REGION Network 49: Phmi Connect
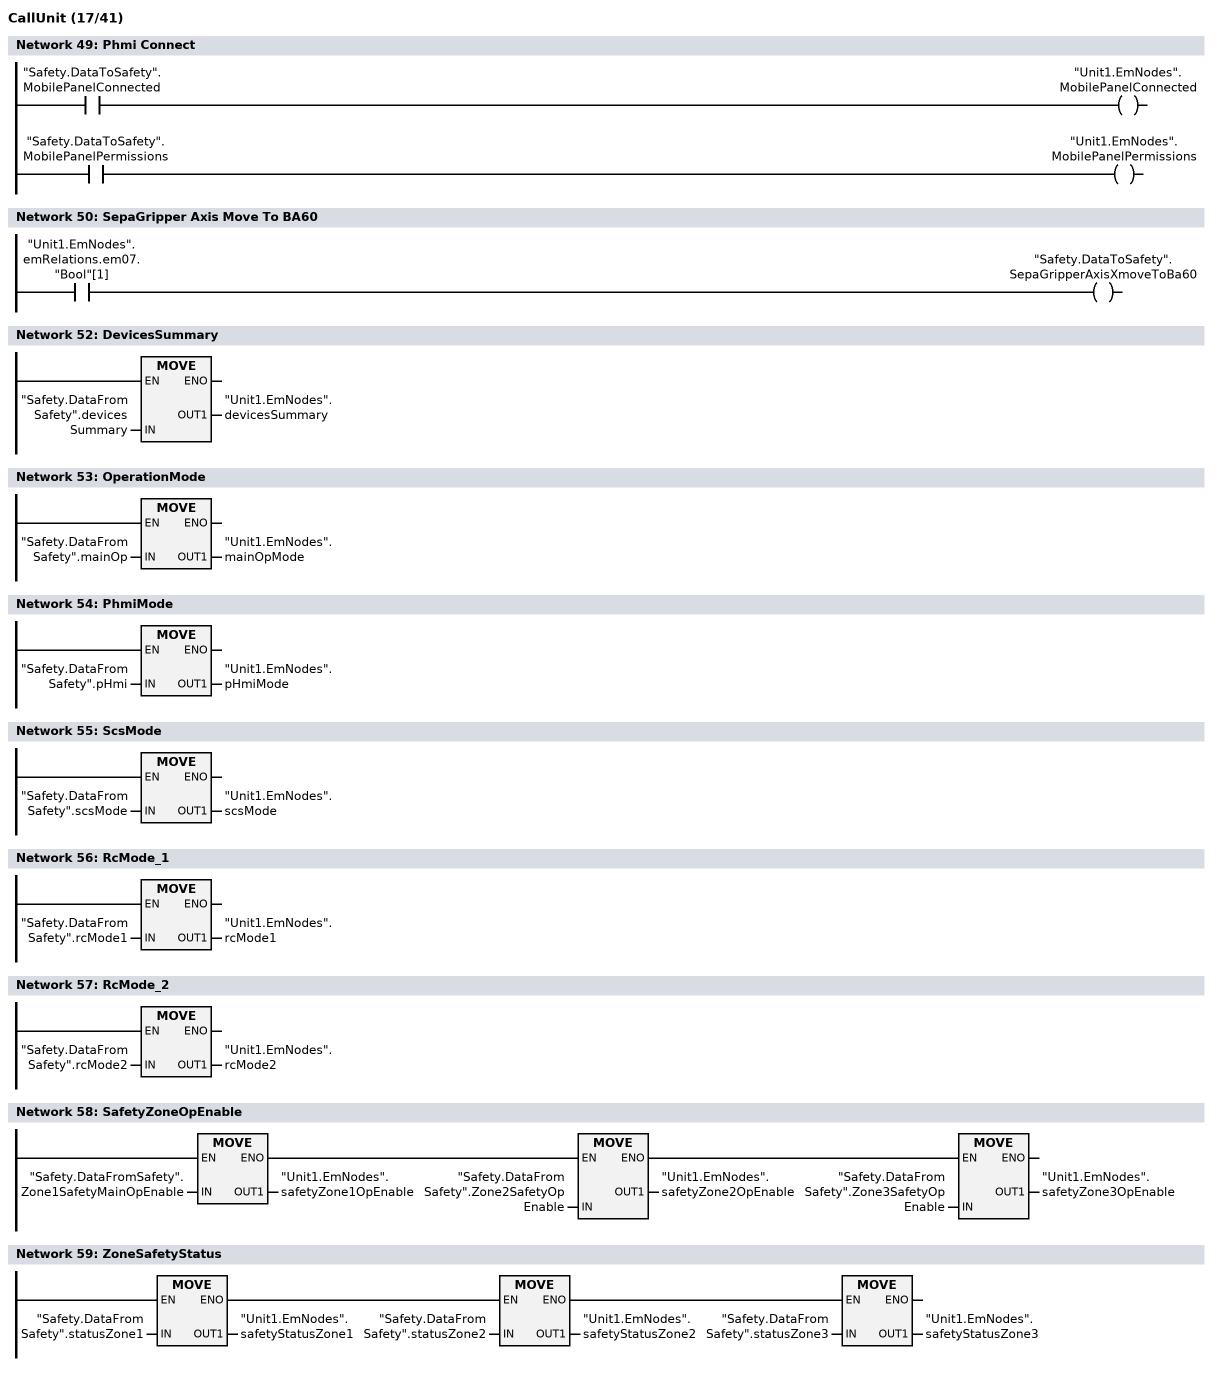
   RUNG wire#powerrail
      Contact( "Safety.DataToSafety".MobilePanelConnected )
      Coil( "Unit1.EmNodes".MobilePanelConnected )
   END_RUNG
   RUNG wire#powerrail
      Contact( "Safety.DataToSafety".MobilePanelPermissions )
      Coil( "Unit1.EmNodes".MobilePanelPermissions )
   END_RUNG
   // the same network as SCL:
   "Unit1.EmNodes".MobilePanelConnected := "Safety.DataToSafety".MobilePanelConnected;
   "Unit1.EmNodes".MobilePanelPermissions := "Safety.DataToSafety".MobilePanelPermissions;
END_REGION

REGION Network 50: SepaGripper Axis Move To BA60
   RUNG wire#powerrail
      Contact( "Unit1.EmNodes".emRelations.em07."Bool"[1] )
      Coil( "Safety.DataToSafety".SepaGripperAxisXmoveToBa60 )
   END_RUNG
   // the same network as SCL:
   "Safety.DataToSafety".SepaGripperAxisXmoveToBa60 := "Unit1.EmNodes".emRelations.em07."Bool"[1];
END_REGION

REGION Network 51: ******************** Data From Safety Mapping ********************
END_REGION

REGION Network 52: DevicesSummary
   RUNG wire#powerrail
      Move(in := "Safety.DataFromSafety".devicesSummary, out1 => "Unit1.EmNodes".devicesSummary)
   END_RUNG
   // the same network as SCL:
   "Unit1.EmNodes".devicesSummary := "Safety.DataFromSafety".devicesSummary;
END_REGION

REGION Network 53: OperationMode
   RUNG wire#powerrail
      Move(in := "Safety.DataFromSafety".mainOp, out1 => "Unit1.EmNodes".mainOpMode)
   END_RUNG
   // the same network as SCL:
   "Unit1.EmNodes".mainOpMode := "Safety.DataFromSafety".mainOp;
END_REGION

REGION Network 54: PhmiMode
   RUNG wire#powerrail
      Move(in := "Safety.DataFromSafety".pHmi, out1 => "Unit1.EmNodes".pHmiMode)
   END_RUNG
   // the same network as SCL:
   "Unit1.EmNodes".pHmiMode := "Safety.DataFromSafety".pHmi;
END_REGION

REGION Network 55: ScsMode
   RUNG wire#powerrail
      Move(in := "Safety.DataFromSafety".scsMode, out1 => "Unit1.EmNodes".scsMode)
   END_RUNG
   // the same network as SCL:
   "Unit1.EmNodes".scsMode := "Safety.DataFromSafety".scsMode;
END_REGION

REGION Network 56: RcMode_1
   RUNG wire#powerrail
      Move(in := "Safety.DataFromSafety".rcMode1, out1 => "Unit1.EmNodes".rcMode1)
   END_RUNG
   // the same network as SCL:
   "Unit1.EmNodes".rcMode1 := "Safety.DataFromSafety".rcMode1;
END_REGION

REGION Network 57: RcMode_2
   RUNG wire#powerrail
      Move(in := "Safety.DataFromSafety".rcMode2, out1 => "Unit1.EmNodes".rcMode2)
   END_RUNG
   // the same network as SCL:
   "Unit1.EmNodes".rcMode2 := "Safety.DataFromSafety".rcMode2;
END_REGION

REGION Network 58: SafetyZoneOpEnable
   RUNG wire#powerrail
      Move(in := "Safety.DataFromSafety".Zone1SafetyMainOpEnable, out1 => "Unit1.EmNodes".safetyZone1OpEnable)
      Move(in := "Safety.DataFromSafety".Zone2SafetyOpEnable, out1 => "Unit1.EmNodes".safetyZone2OpEnable)
      Move(in := "Safety.DataFromSafety".Zone3SafetyOpEnable, out1 => "Unit1.EmNodes".safetyZone3OpEnable)
   END_RUNG
   // the same network as SCL:
   "Unit1.EmNodes".safetyZone1OpEnable := "Safety.DataFromSafety".Zone1SafetyMainOpEnable;
   "Unit1.EmNodes".safetyZone2OpEnable := "Safety.DataFromSafety".Zone2SafetyOpEnable;
   "Unit1.EmNodes".safetyZone3OpEnable := "Safety.DataFromSafety".Zone3SafetyOpEnable;
END_REGION

REGION Network 59: ZoneSafetyStatus
   RUNG wire#powerrail
      Move(in := "Safety.DataFromSafety".statusZone1, out1 => "Unit1.EmNodes".safetyStatusZone1)
      Move(in := "Safety.DataFromSafety".statusZone2, out1 => "Unit1.EmNodes".safetyStatusZone2)
      Move(in := "Safety.DataFromSafety".statusZone3, out1 => "Unit1.EmNodes".safetyStatusZone3)
   END_RUNG
   // the same network as SCL:
   "Unit1.EmNodes".safetyStatusZone1 := "Safety.DataFromSafety".statusZone1;
   "Unit1.EmNodes".safetyStatusZone2 := "Safety.DataFromSafety".statusZone2;
   "Unit1.EmNodes".safetyStatusZone3 := "Safety.DataFromSafety".statusZone3;
END_REGION

REGION Network 60: SafetySensor
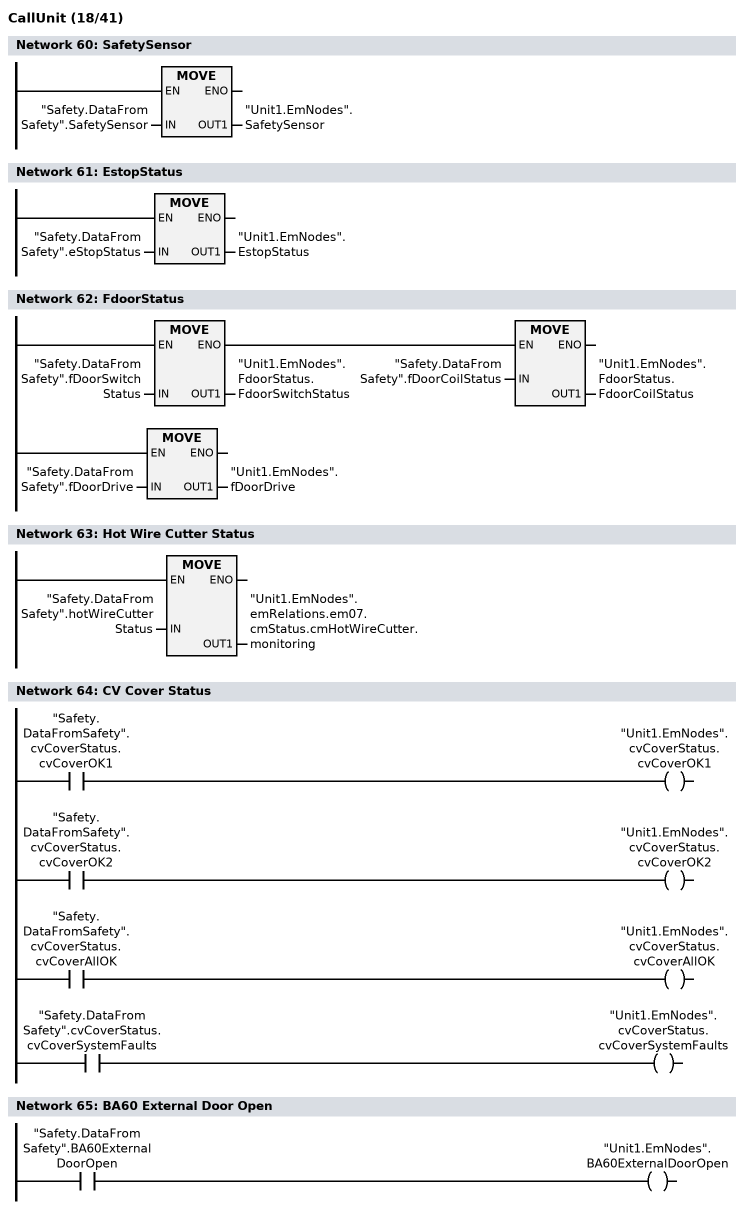
   RUNG wire#powerrail
      Move(in := "Safety.DataFromSafety".SafetySensor, out1 => "Unit1.EmNodes".SafetySensor)
   END_RUNG
   // the same network as SCL:
   "Unit1.EmNodes".SafetySensor := "Safety.DataFromSafety".SafetySensor;
END_REGION

REGION Network 61: EstopStatus
   RUNG wire#powerrail
      Move(in := "Safety.DataFromSafety".eStopStatus, out1 => "Unit1.EmNodes".EstopStatus)
   END_RUNG
   // the same network as SCL:
   "Unit1.EmNodes".EstopStatus := "Safety.DataFromSafety".eStopStatus;
END_REGION

REGION Network 62: FdoorStatus
   RUNG wire#powerrail
      Move(in := "Safety.DataFromSafety".fDoorSwitchStatus, out1 => "Unit1.EmNodes".FdoorStatus.FdoorSwitchStatus)
      Move(in := "Safety.DataFromSafety".fDoorCoilStatus, out1 => "Unit1.EmNodes".FdoorStatus.FdoorCoilStatus)
   END_RUNG
   RUNG wire#powerrail
      Move(in := "Safety.DataFromSafety".fDoorDrive, out1 => "Unit1.EmNodes".fDoorDrive)
   END_RUNG
   // the same network as SCL:
   "Unit1.EmNodes".FdoorStatus.FdoorSwitchStatus := "Safety.DataFromSafety".fDoorSwitchStatus;
   "Unit1.EmNodes".FdoorStatus.FdoorCoilStatus := "Safety.DataFromSafety".fDoorCoilStatus;
   "Unit1.EmNodes".fDoorDrive := "Safety.DataFromSafety".fDoorDrive;
END_REGION

REGION Network 63: Hot Wire Cutter Status
   RUNG wire#powerrail
      Move(in := "Safety.DataFromSafety".hotWireCutterStatus, out1 => "Unit1.EmNodes".emRelations.em07.cmStatus.cmHotWireCutter.monitoring)
   END_RUNG
   // the same network as SCL:
   "Unit1.EmNodes".emRelations.em07.cmStatus.cmHotWireCutter.monitoring := "Safety.DataFromSafety".hotWireCutterStatus;
END_REGION

REGION Network 64: CV Cover Status
   RUNG wire#powerrail
      Contact( "Safety.DataFromSafety".cvCoverStatus.cvCoverOK1 )
      Coil( "Unit1.EmNodes".cvCoverStatus.cvCoverOK1 )
   END_RUNG
   RUNG wire#powerrail
      Contact( "Safety.DataFromSafety".cvCoverStatus.cvCoverOK2 )
      Coil( "Unit1.EmNodes".cvCoverStatus.cvCoverOK2 )
   END_RUNG
   RUNG wire#powerrail
      Contact( "Safety.DataFromSafety".cvCoverStatus.cvCoverAllOK )
      Coil( "Unit1.EmNodes".cvCoverStatus.cvCoverAllOK )
   END_RUNG
   RUNG wire#powerrail
      Contact( "Safety.DataFromSafety".cvCoverStatus.cvCoverSystemFaults )
      Coil( "Unit1.EmNodes".cvCoverStatus.cvCoverSystemFaults )
   END_RUNG
   // the same network as SCL:
   "Unit1.EmNodes".cvCoverStatus.cvCoverOK1 := "Safety.DataFromSafety".cvCoverStatus.cvCoverOK1;
   "Unit1.EmNodes".cvCoverStatus.cvCoverOK2 := "Safety.DataFromSafety".cvCoverStatus.cvCoverOK2;
   "Unit1.EmNodes".cvCoverStatus.cvCoverAllOK := "Safety.DataFromSafety".cvCoverStatus.cvCoverAllOK;
   "Unit1.EmNodes".cvCoverStatus.cvCoverSystemFaults := "Safety.DataFromSafety".cvCoverStatus.cvCoverSystemFaults;
END_REGION

REGION Network 65: BA60 External Door Open
   RUNG wire#powerrail
      Contact( "Safety.DataFromSafety".BA60ExternalDoorOpen )
      Coil( "Unit1.EmNodes".BA60ExternalDoorOpen )
   END_RUNG
   // the same network as SCL:
   "Unit1.EmNodes".BA60ExternalDoorOpen := "Safety.DataFromSafety".BA60ExternalDoorOpen;
END_REGION

REGION Network 66: All SF Door Open
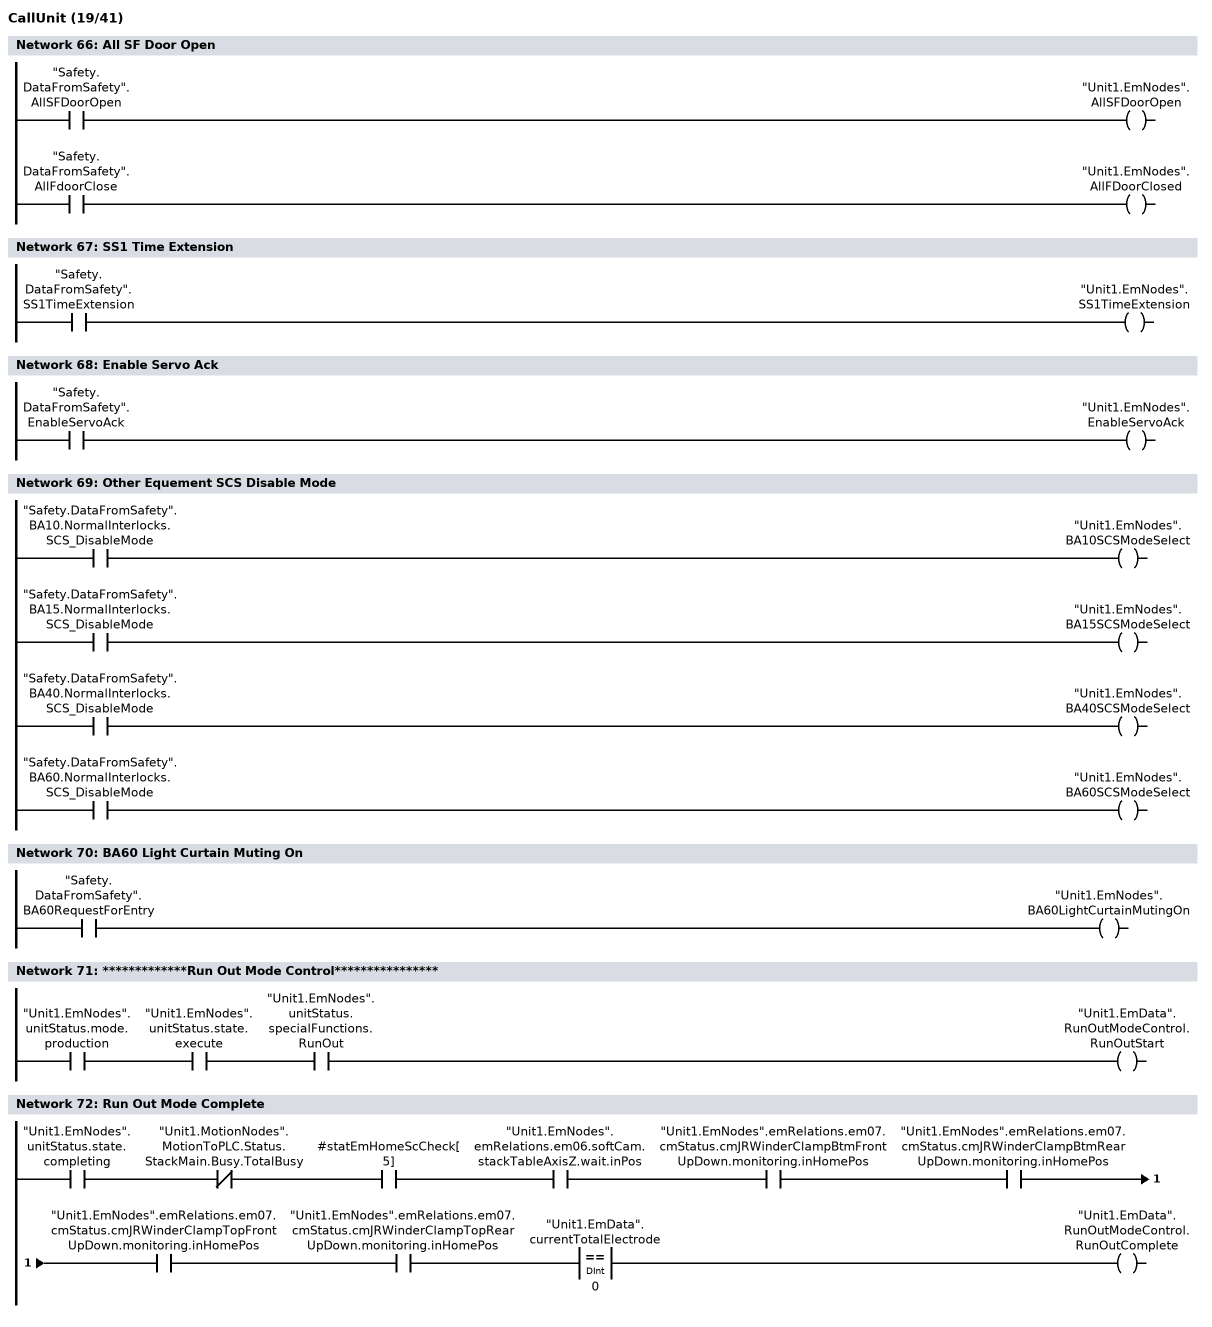
   RUNG wire#powerrail
      Contact( "Safety.DataFromSafety".AllSFDoorOpen )
      Coil( "Unit1.EmNodes".AllSFDoorOpen )
   END_RUNG
   RUNG wire#powerrail
      Contact( "Safety.DataFromSafety".AllFdoorClose )
      Coil( "Unit1.EmNodes".AllFDoorClosed )
   END_RUNG
   // the same network as SCL:
   "Unit1.EmNodes".AllSFDoorOpen := "Safety.DataFromSafety".AllSFDoorOpen;
   "Unit1.EmNodes".AllFDoorClosed := "Safety.DataFromSafety".AllFdoorClose;
END_REGION

REGION Network 67: SS1 Time Extension
   RUNG wire#powerrail
      Contact( "Safety.DataFromSafety".SS1TimeExtension )
      Coil( "Unit1.EmNodes".SS1TimeExtension )
   END_RUNG
   // the same network as SCL:
   "Unit1.EmNodes".SS1TimeExtension := "Safety.DataFromSafety".SS1TimeExtension;
END_REGION

REGION Network 68: Enable Servo Ack
   RUNG wire#powerrail
      Contact( "Safety.DataFromSafety".EnableServoAck )
      Coil( "Unit1.EmNodes".EnableServoAck )
   END_RUNG
   // the same network as SCL:
   "Unit1.EmNodes".EnableServoAck := "Safety.DataFromSafety".EnableServoAck;
END_REGION

REGION Network 69: Other Equement SCS Disable Mode
   RUNG wire#powerrail
      Contact( "Safety.DataFromSafety".BA10.NormalInterlocks.SCS_DisableMode )
      Coil( "Unit1.EmNodes".BA10SCSModeSelect )
   END_RUNG
   RUNG wire#powerrail
      Contact( "Safety.DataFromSafety".BA15.NormalInterlocks.SCS_DisableMode )
      Coil( "Unit1.EmNodes".BA15SCSModeSelect )
   END_RUNG
   RUNG wire#powerrail
      Contact( "Safety.DataFromSafety".BA40.NormalInterlocks.SCS_DisableMode )
      Coil( "Unit1.EmNodes".BA40SCSModeSelect )
   END_RUNG
   RUNG wire#powerrail
      Contact( "Safety.DataFromSafety".BA60.NormalInterlocks.SCS_DisableMode )
      Coil( "Unit1.EmNodes".BA60SCSModeSelect )
   END_RUNG
   // the same network as SCL:
   "Unit1.EmNodes".BA10SCSModeSelect := "Safety.DataFromSafety".BA10.NormalInterlocks.SCS_DisableMode;
   "Unit1.EmNodes".BA15SCSModeSelect := "Safety.DataFromSafety".BA15.NormalInterlocks.SCS_DisableMode;
   "Unit1.EmNodes".BA40SCSModeSelect := "Safety.DataFromSafety".BA40.NormalInterlocks.SCS_DisableMode;
   "Unit1.EmNodes".BA60SCSModeSelect := "Safety.DataFromSafety".BA60.NormalInterlocks.SCS_DisableMode;
END_REGION

REGION Network 70: BA60 Light Curtain Muting On
   RUNG wire#powerrail
      Contact( "Safety.DataFromSafety".BA60RequestForEntry )
      Coil( "Unit1.EmNodes".BA60LightCurtainMutingOn )
   END_RUNG
   // the same network as SCL:
   "Unit1.EmNodes".BA60LightCurtainMutingOn := "Safety.DataFromSafety".BA60RequestForEntry;
END_REGION

REGION Network 71: *************Run Out Mode Control****************
   RUNG wire#powerrail
      Contact( "Unit1.EmNodes".unitStatus.mode.production )
      Contact( "Unit1.EmNodes".unitStatus.state.execute )
      Contact( "Unit1.EmNodes".unitStatus.specialFunctions.RunOut )
      Coil( "Unit1.EmData".RunOutModeControl.RunOutStart )
   END_RUNG
   // the same network as SCL:
   "Unit1.EmData".RunOutModeControl.RunOutStart := "Unit1.EmNodes".unitStatus.mode.production AND "Unit1.EmNodes".unitStatus.state.execute AND "Unit1.EmNodes".unitStatus.specialFunctions.RunOut;
END_REGION

REGION Network 72: Run Out Mode Complete
   RUNG wire#powerrail
      Contact( "Unit1.EmNodes".unitStatus.state.completing )
      I_Contact( "Unit1.MotionNodes".MotionToPLC.Status.StackMain.Busy.TotalBusy )
      Contact( #statEmHomeScCheck[5] )
      Contact( "Unit1.EmNodes".emRelations.em06.softCam.stackTableAxisZ.wait.inPos )
      Contact( "Unit1.EmNodes".emRelations.em07.cmStatus.cmJRWinderClampBtmFrontUpDown.monitoring.inHomePos )
      Contact( "Unit1.EmNodes".emRelations.em07.cmStatus.cmJRWinderClampBtmRearUpDown.monitoring.inHomePos )
      Contact( "Unit1.EmNodes".emRelations.em07.cmStatus.cmJRWinderClampTopFrontUpDown.monitoring.inHomePos )
      Contact( "Unit1.EmNodes".emRelations.em07.cmStatus.cmJRWinderClampTopRearUpDown.monitoring.inHomePos )
      { S7_Templates := "SrcType := DInt" } EQ_Contact(in1 := "Unit1.EmData".currentTotalElectrode, in2 := 0)
      Coil( "Unit1.EmData".RunOutModeControl.RunOutComplete )
   END_RUNG
   // the same network as SCL:
   "Unit1.EmData".RunOutModeControl.RunOutComplete := "Unit1.EmNodes".unitStatus.state.completing AND NOT "Unit1.MotionNodes".MotionToPLC.Status.StackMain.Busy.TotalBusy AND #statEmHomeScCheck[5] AND "Unit1.EmNodes".emRelations.em06.softCam.stackTableAxisZ.wait.inPos AND "Unit1.EmNodes".emRelations.em07.cmStatus.cmJRWinderClampBtmFrontUpDown.monitoring.inHomePos AND "Unit1.EmNodes".emRelations.em07.cmStatus.cmJRWinderClampBtmRearUpDown.monitoring.inHomePos AND "Unit1.EmNodes".emRelations.em07.cmStatus.cmJRWinderClampTopFrontUpDown.monitoring.inHomePos AND "Unit1.EmNodes".emRelations.em07.cmStatus.cmJRWinderClampTopRearUpDown.monitoring.inHomePos AND ("Unit1.EmData".currentTotalElectrode = 0);
END_REGION

REGION Network 73: ******************** FAT Mode ********************
END_REGION

REGION Network 74: HoursTest Mode
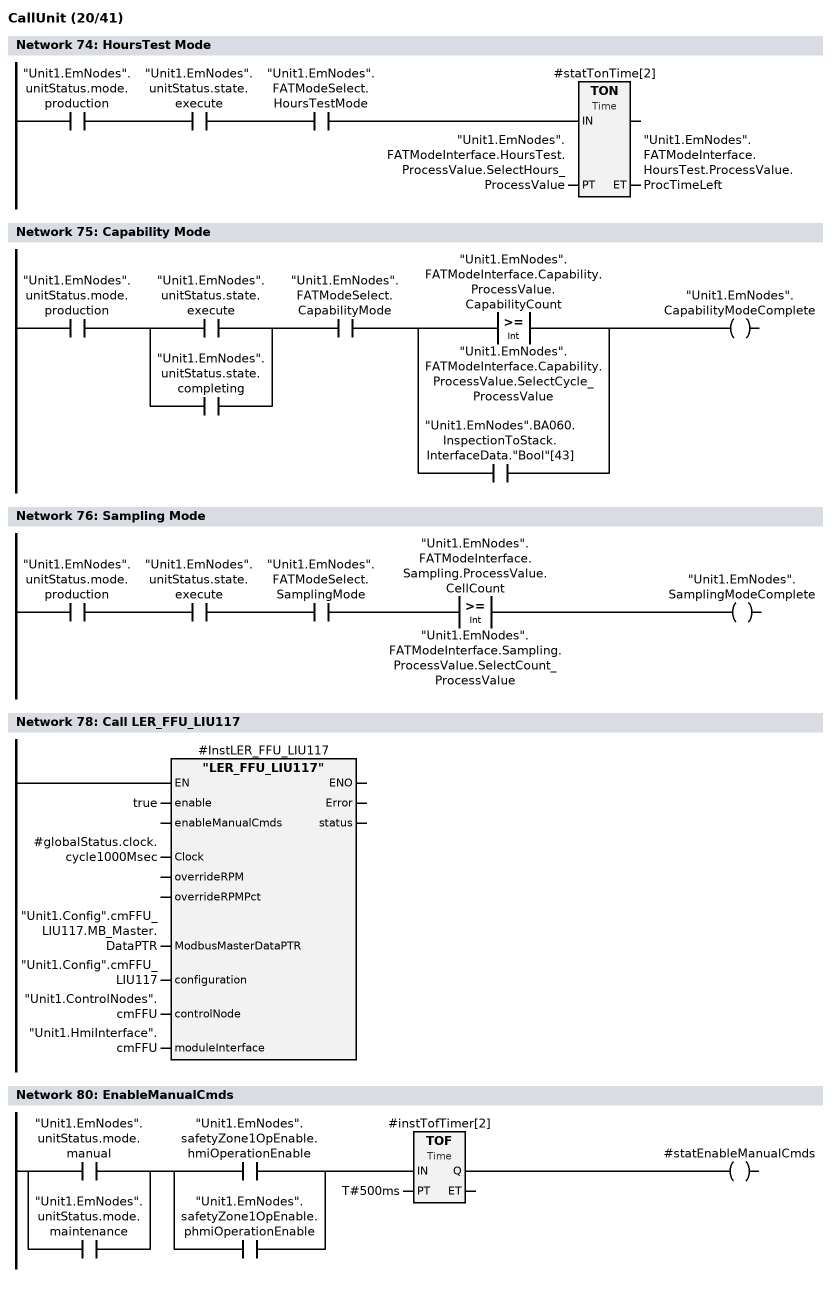
   RUNG wire#powerrail
      Contact( "Unit1.EmNodes".unitStatus.mode.production )
      Contact( "Unit1.EmNodes".unitStatus.state.execute )
      Contact( "Unit1.EmNodes".FATModeSelect.HoursTestMode )
      { S7_Templates := "time_type := Time" } #statTonTime[2].TON(pt := "Unit1.EmNodes".FATModeInterface.HoursTest.ProcessValue.SelectHours_ProcessValue, et => "Unit1.EmNodes".FATModeInterface.HoursTest.ProcessValue.ProcTimeLeft)
   END_RUNG
   // the same network as SCL:
   #statTonTime[2].TON(IN := "Unit1.EmNodes".unitStatus.mode.production AND "Unit1.EmNodes".unitStatus.state.execute AND "Unit1.EmNodes".FATModeSelect.HoursTestMode,
                       PT := "Unit1.EmNodes".FATModeInterface.HoursTest.ProcessValue.SelectHours_ProcessValue,
                       ET => "Unit1.EmNodes".FATModeInterface.HoursTest.ProcessValue.ProcTimeLeft);
END_REGION

REGION Network 75: Capability Mode
   RUNG wire#powerrail
      Contact( "Unit1.EmNodes".unitStatus.mode.production )
      wire#w1
      Contact( "Unit1.EmNodes".unitStatus.state.execute )
      wire#w2
      Contact( "Unit1.EmNodes".FATModeSelect.CapabilityMode )
      wire#w3
      { S7_Templates := "SrcType := Int" } GE_Contact(in1 := "Unit1.EmNodes".FATModeInterface.Capability.ProcessValue.CapabilityCount, in2 := "Unit1.EmNodes".FATModeInterface.Capability.ProcessValue.SelectCycle_ProcessValue)
      wire#w4
      Coil( "Unit1.EmNodes".CapabilityModeComplete )
   END_RUNG
   RUNG wire#w1
      Contact( "Unit1.EmNodes".unitStatus.state.completing )
   END_RUNG wire#w2
   RUNG wire#w3
      Contact( "Unit1.EmNodes".BA060.InspectionToStack.InterfaceData."Bool"[43] )
   END_RUNG wire#w4
   // the same network as SCL:
   "Unit1.EmNodes".CapabilityModeComplete := "Unit1.EmNodes".unitStatus.mode.production AND ("Unit1.EmNodes".unitStatus.state.execute OR "Unit1.EmNodes".unitStatus.state.completing) AND "Unit1.EmNodes".FATModeSelect.CapabilityMode AND (("Unit1.EmNodes".FATModeInterface.Capability.ProcessValue.CapabilityCount >= "Unit1.EmNodes".FATModeInterface.Capability.ProcessValue.SelectCycle_ProcessValue) OR "Unit1.EmNodes".BA060.InspectionToStack.InterfaceData."Bool"[43]);
END_REGION

REGION Network 76: Sampling Mode
   RUNG wire#powerrail
      Contact( "Unit1.EmNodes".unitStatus.mode.production )
      Contact( "Unit1.EmNodes".unitStatus.state.execute )
      Contact( "Unit1.EmNodes".FATModeSelect.SamplingMode )
      { S7_Templates := "SrcType := Int" } GE_Contact(in1 := "Unit1.EmNodes".FATModeInterface.Sampling.ProcessValue.CellCount, in2 := "Unit1.EmNodes".FATModeInterface.Sampling.ProcessValue.SelectCount_ProcessValue)
      Coil( "Unit1.EmNodes".SamplingModeComplete )
   END_RUNG
   // the same network as SCL:
   "Unit1.EmNodes".SamplingModeComplete := "Unit1.EmNodes".unitStatus.mode.production AND "Unit1.EmNodes".unitStatus.state.execute AND "Unit1.EmNodes".FATModeSelect.SamplingMode AND ("Unit1.EmNodes".FATModeInterface.Sampling.ProcessValue.CellCount >= "Unit1.EmNodes".FATModeInterface.Sampling.ProcessValue.SelectCount_ProcessValue);
END_REGION

REGION Network 77: *************** FFU LIU117 (MCU) ***************************
END_REGION

REGION Network 78: Call LER_FFU_LIU117
   RUNG wire#powerrail
      #InstLER_FFU_LIU117(enable := true, enableManualCmds :=, Clock := #globalStatus.clock.cycle1000Msec, overrideRPM :=, overrideRPMPct :=, ModbusMasterDataPTR := "Unit1.Config".cmFFU_LIU117.MB_Master.DataPTR, configuration := "Unit1.Config".cmFFU_LIU117, controlNode := "Unit1.ControlNodes".cmFFU, moduleInterface := "Unit1.HmiInterface".cmFFU, Error =>, status =>)
   END_RUNG
   // the same network as SCL:
   #InstLER_FFU_LIU117(enable := true,   // "LER_FFU_LIU117"
                       Clock := #globalStatus.clock.cycle1000Msec,
                       ModbusMasterDataPTR := "Unit1.Config".cmFFU_LIU117.MB_Master.DataPTR,
                       configuration := "Unit1.Config".cmFFU_LIU117,
                       controlNode := "Unit1.ControlNodes".cmFFU,
                       moduleInterface := "Unit1.HmiInterface".cmFFU);
END_REGION

REGION Network 79: ******************** Brake Test ********************
END_REGION

REGION Network 80: EnableManualCmds
   RUNG wire#powerrail
      Contact( "Unit1.EmNodes".unitStatus.mode.manual )
      wire#w1
      Contact( "Unit1.EmNodes".safetyZone1OpEnable.hmiOperationEnable )
      wire#w2
      { S7_Templates := "time_type := Time" } #instTofTimer[2].TOF(pt := T#500ms, et =>)
      Coil( #statEnableManualCmds )
   END_RUNG
   RUNG wire#powerrail
      Contact( "Unit1.EmNodes".unitStatus.mode.maintenance )
   END_RUNG wire#w1
   RUNG wire#w1
      Contact( "Unit1.EmNodes".safetyZone1OpEnable.phmiOperationEnable )
   END_RUNG wire#w2
   // the same network as SCL:
   #instTofTimer[2].TOF(IN := ("Unit1.EmNodes".unitStatus.mode.manual OR "Unit1.EmNodes".unitStatus.mode.maintenance) AND ("Unit1.EmNodes".safetyZone1OpEnable.hmiOperationEnable OR "Unit1.EmNodes".safetyZone1OpEnable.phmiOperationEnable),
                        PT := T#500ms);
   #statEnableManualCmds := #instTofTimer[2].Q;
END_REGION

REGION Network 81: All Brake Test Error
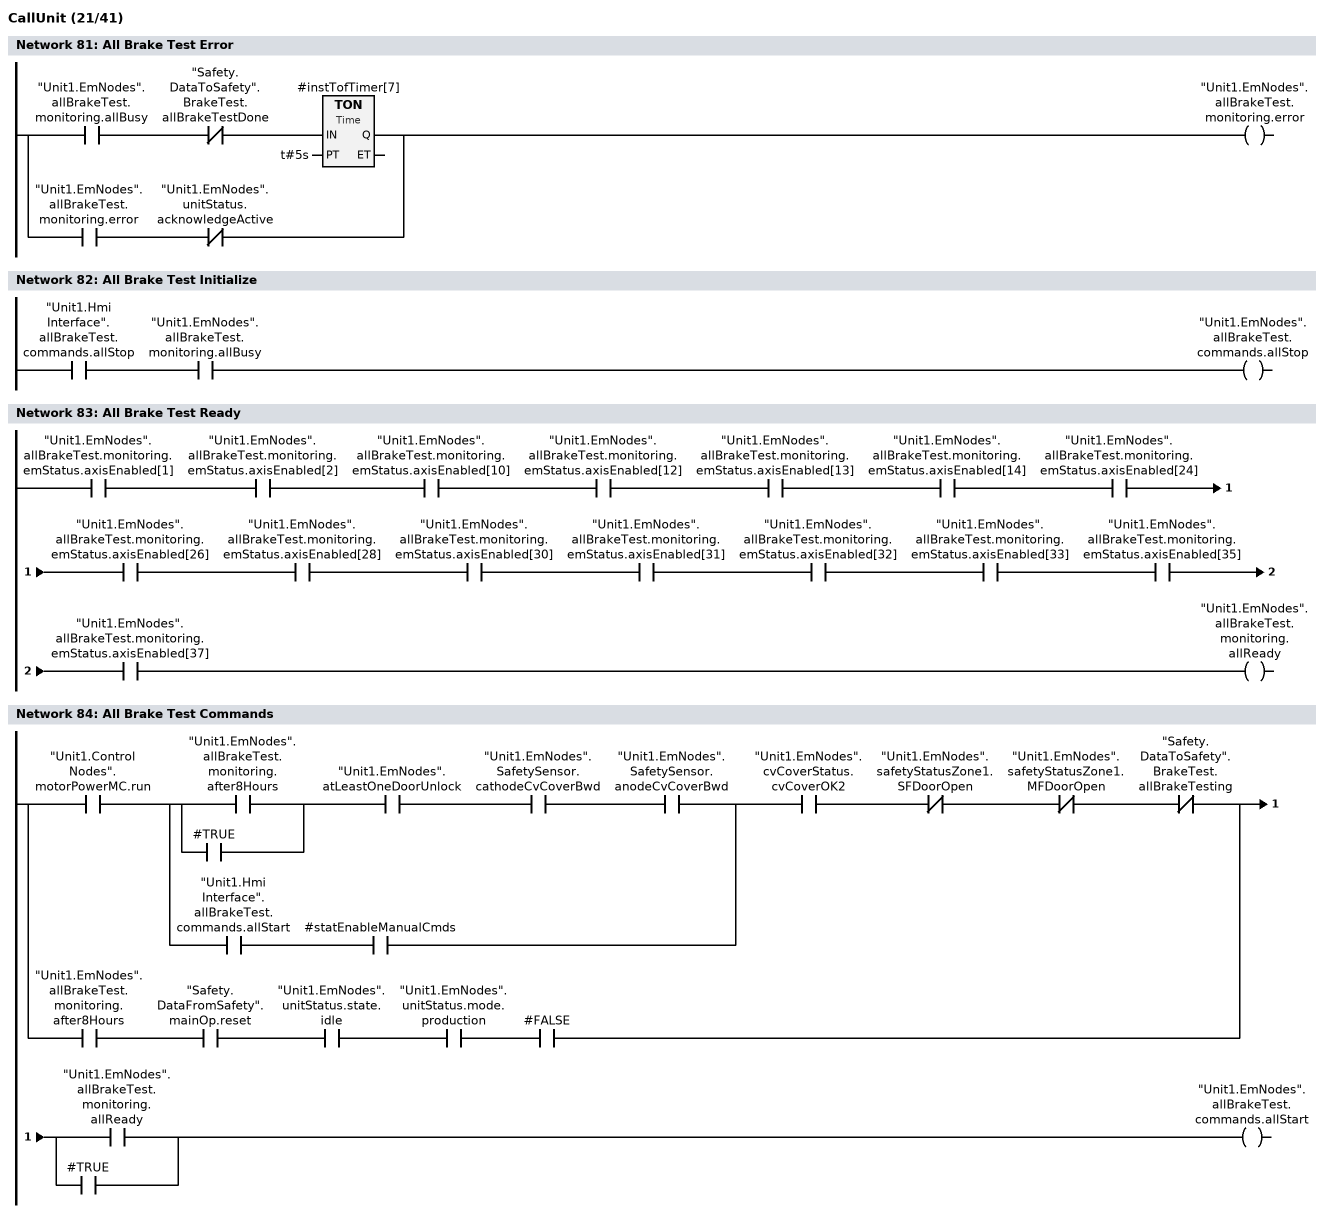
   RUNG wire#powerrail
      Contact( "Unit1.EmNodes".allBrakeTest.monitoring.allBusy )
      I_Contact( "Safety.DataToSafety".BrakeTest.allBrakeTestDone )
      { S7_Templates := "time_type := Time" } #instTofTimer[7].TON(pt := t#5s, et =>)
      wire#w1
      Coil( "Unit1.EmNodes".allBrakeTest.monitoring.error )
   END_RUNG
   RUNG wire#powerrail
      Contact( "Unit1.EmNodes".allBrakeTest.monitoring.error )
      I_Contact( "Unit1.EmNodes".unitStatus.acknowledgeActive )
   END_RUNG wire#w1
   // the same network as SCL:
   #instTofTimer[7].TON(IN := "Unit1.EmNodes".allBrakeTest.monitoring.allBusy AND NOT "Safety.DataToSafety".BrakeTest.allBrakeTestDone,
                        PT := t#5s);
   "Unit1.EmNodes".allBrakeTest.monitoring.error := #instTofTimer[7].Q OR ("Unit1.EmNodes".allBrakeTest.monitoring.error AND NOT "Unit1.EmNodes".unitStatus.acknowledgeActive);
END_REGION

REGION Network 82: All Brake Test Initialize
   RUNG wire#powerrail
      Contact( "Unit1.HmiInterface".allBrakeTest.commands.allStop )
      Contact( "Unit1.EmNodes".allBrakeTest.monitoring.allBusy )
      Coil( "Unit1.EmNodes".allBrakeTest.commands.allStop )
   END_RUNG
   // the same network as SCL:
   "Unit1.EmNodes".allBrakeTest.commands.allStop := "Unit1.HmiInterface".allBrakeTest.commands.allStop AND "Unit1.EmNodes".allBrakeTest.monitoring.allBusy;
END_REGION

REGION Network 83: All Brake Test Ready
   RUNG wire#powerrail
      Contact( "Unit1.EmNodes".allBrakeTest.monitoring.emStatus.axisEnabled[1] )
      Contact( "Unit1.EmNodes".allBrakeTest.monitoring.emStatus.axisEnabled[2] )
      Contact( "Unit1.EmNodes".allBrakeTest.monitoring.emStatus.axisEnabled[10] )
      Contact( "Unit1.EmNodes".allBrakeTest.monitoring.emStatus.axisEnabled[12] )
      Contact( "Unit1.EmNodes".allBrakeTest.monitoring.emStatus.axisEnabled[13] )
      Contact( "Unit1.EmNodes".allBrakeTest.monitoring.emStatus.axisEnabled[14] )
      Contact( "Unit1.EmNodes".allBrakeTest.monitoring.emStatus.axisEnabled[24] )
      Contact( "Unit1.EmNodes".allBrakeTest.monitoring.emStatus.axisEnabled[26] )
      Contact( "Unit1.EmNodes".allBrakeTest.monitoring.emStatus.axisEnabled[28] )
      Contact( "Unit1.EmNodes".allBrakeTest.monitoring.emStatus.axisEnabled[30] )
      Contact( "Unit1.EmNodes".allBrakeTest.monitoring.emStatus.axisEnabled[31] )
      Contact( "Unit1.EmNodes".allBrakeTest.monitoring.emStatus.axisEnabled[32] )
      Contact( "Unit1.EmNodes".allBrakeTest.monitoring.emStatus.axisEnabled[33] )
      Contact( "Unit1.EmNodes".allBrakeTest.monitoring.emStatus.axisEnabled[35] )
      Contact( "Unit1.EmNodes".allBrakeTest.monitoring.emStatus.axisEnabled[37] )
      Coil( "Unit1.EmNodes".allBrakeTest.monitoring.allReady )
   END_RUNG
   // the same network as SCL:
   "Unit1.EmNodes".allBrakeTest.monitoring.allReady := "Unit1.EmNodes".allBrakeTest.monitoring.emStatus.axisEnabled[1] AND "Unit1.EmNodes".allBrakeTest.monitoring.emStatus.axisEnabled[2] AND "Unit1.EmNodes".allBrakeTest.monitoring.emStatus.axisEnabled[10] AND "Unit1.EmNodes".allBrakeTest.monitoring.emStatus.axisEnabled[12] AND "Unit1.EmNodes".allBrakeTest.monitoring.emStatus.axisEnabled[13] AND "Unit1.EmNodes".allBrakeTest.monitoring.emStatus.axisEnabled[14] AND "Unit1.EmNodes".allBrakeTest.monitoring.emStatus.axisEnabled[24] AND "Unit1.EmNodes".allBrakeTest.monitoring.emStatus.axisEnabled[26] AND "Unit1.EmNodes".allBrakeTest.monitoring.emStatus.axisEnabled[28] AND "Unit1.EmNodes".allBrakeTest.monitoring.emStatus.axisEnabled[30] AND "Unit1.EmNodes".allBrakeTest.monitoring.emStatus.axisEnabled[31] AND "Unit1.EmNodes".allBrakeTest.monitoring.emStatus.axisEnabled[32] AND "Unit1.EmNodes".allBrakeTest.monitoring.emStatus.axisEnabled[33] AND "Unit1.EmNodes".allBrakeTest.monitoring.emStatus.axisEnabled[35] AND "Unit1.EmNodes".allBrakeTest.monitoring.emStatus.axisEnabled[37];
END_REGION

REGION Network 84: All Brake Test Commands
   RUNG wire#powerrail
      Contact( "Unit1.ControlNodes".motorPowerMC.run )
      wire#w1
      Contact( "Unit1.EmNodes".allBrakeTest.monitoring.after8Hours )
      wire#w2
      Contact( "Unit1.EmNodes".atLeastOneDoorUnlock )
      Contact( "Unit1.EmNodes".SafetySensor.cathodeCvCoverBwd )
      Contact( "Unit1.EmNodes".SafetySensor.anodeCvCoverBwd )
      wire#w3
      Contact( "Unit1.EmNodes".cvCoverStatus.cvCoverOK2 )
      I_Contact( "Unit1.EmNodes".safetyStatusZone1.SFDoorOpen )
      I_Contact( "Unit1.EmNodes".safetyStatusZone1.MFDoorOpen )
      I_Contact( "Safety.DataToSafety".BrakeTest.allBrakeTesting )
      wire#w4
      Contact( "Unit1.EmNodes".allBrakeTest.monitoring.allReady )
      wire#w5
      Coil( "Unit1.EmNodes".allBrakeTest.commands.allStart )
   END_RUNG
   RUNG wire#w1
      Contact( #TRUE )
   END_RUNG wire#w2
   RUNG wire#w1
      Contact( "Unit1.HmiInterface".allBrakeTest.commands.allStart )
      Contact( #statEnableManualCmds )
   END_RUNG wire#w3
   RUNG wire#powerrail
      Contact( "Unit1.EmNodes".allBrakeTest.monitoring.after8Hours )
      Contact( "Safety.DataFromSafety".mainOp.reset )
      Contact( "Unit1.EmNodes".unitStatus.state.idle )
      Contact( "Unit1.EmNodes".unitStatus.mode.production )
      Contact( #FALSE )
   END_RUNG wire#w4
   RUNG wire#w4
      Contact( #TRUE )
   END_RUNG wire#w5
   // the same network as SCL:
   "Unit1.EmNodes".allBrakeTest.commands.allStart := (("Unit1.ControlNodes".motorPowerMC.run AND ((("Unit1.EmNodes".allBrakeTest.monitoring.after8Hours OR #TRUE) AND "Unit1.EmNodes".atLeastOneDoorUnlock AND "Unit1.EmNodes".SafetySensor.cathodeCvCoverBwd AND "Unit1.EmNodes".SafetySensor.anodeCvCoverBwd) OR ("Unit1.HmiInterface".allBrakeTest.commands.allStart AND #statEnableManualCmds)) AND "Unit1.EmNodes".cvCoverStatus.cvCoverOK2 AND NOT "Unit1.EmNodes".safetyStatusZone1.SFDoorOpen AND NOT "Unit1.EmNodes".safetyStatusZone1.MFDoorOpen AND NOT "Safety.DataToSafety".BrakeTest.allBrakeTesting) OR ("Unit1.EmNodes".allBrakeTest.monitoring.after8Hours AND "Safety.DataFromSafety".mainOp.reset AND "Unit1.EmNodes".unitStatus.state.idle AND "Unit1.EmNodes".unitStatus.mode.production AND #FALSE)) AND ("Unit1.EmNodes".allBrakeTest.monitoring.allReady OR #TRUE);
END_REGION

REGION Network 85: Em Brake Test Status Summary
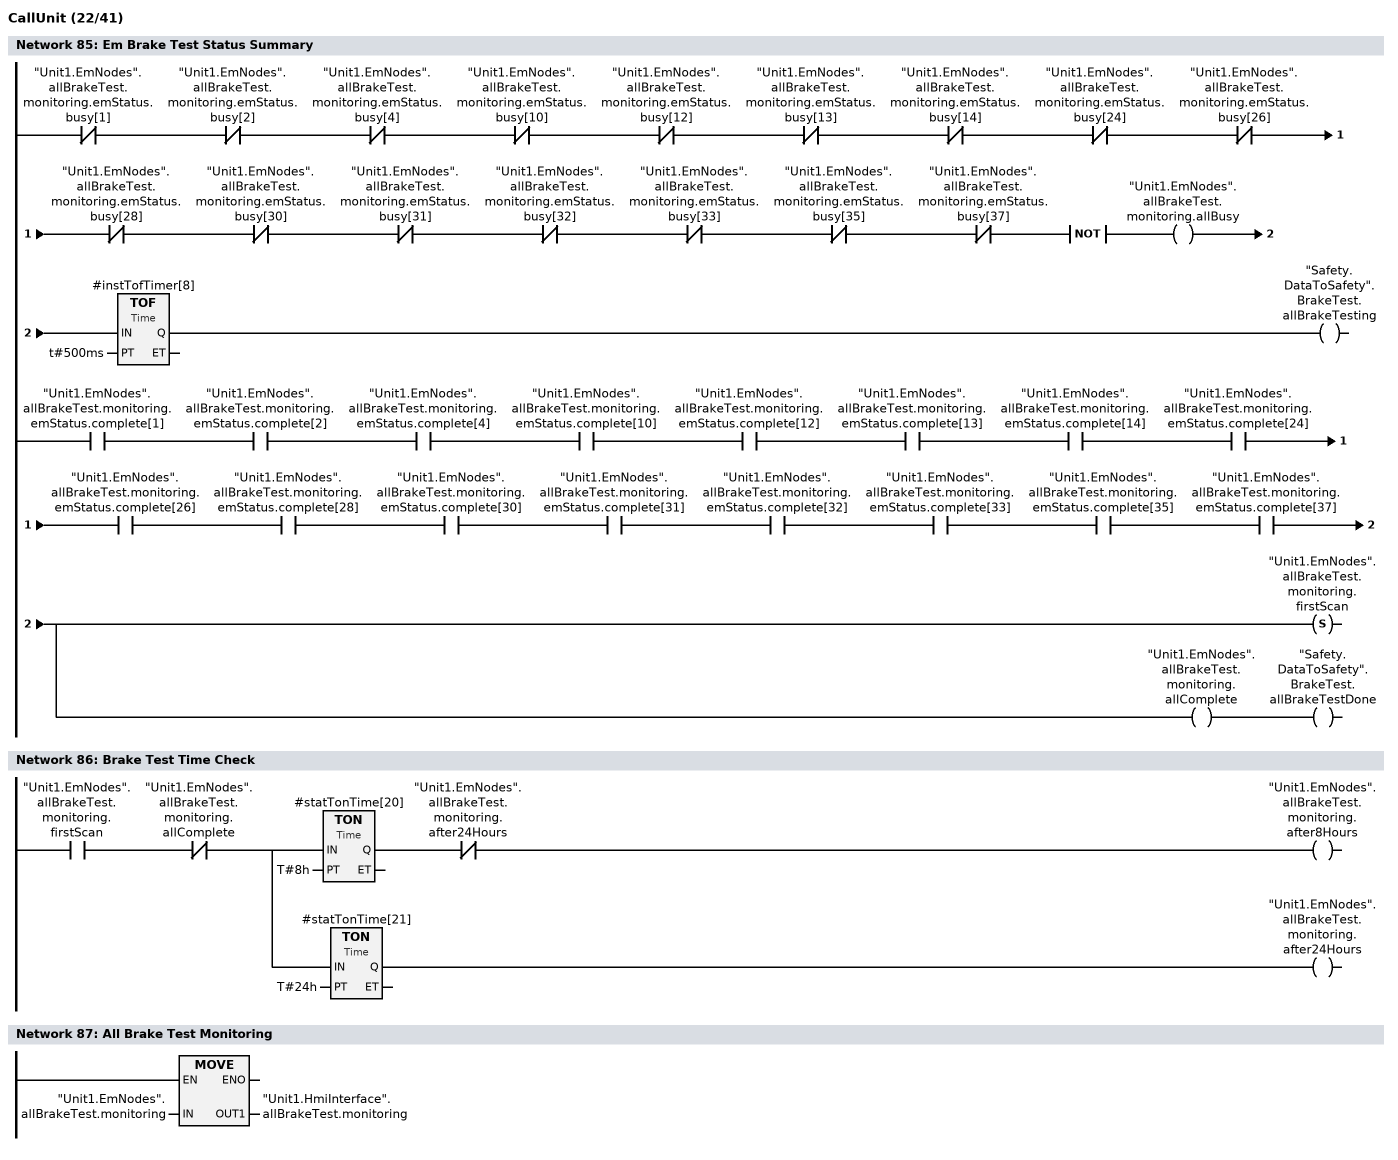
   RUNG wire#powerrail
      I_Contact( "Unit1.EmNodes".allBrakeTest.monitoring.emStatus.busy[1] )
      I_Contact( "Unit1.EmNodes".allBrakeTest.monitoring.emStatus.busy[2] )
      I_Contact( "Unit1.EmNodes".allBrakeTest.monitoring.emStatus.busy[4] )
      I_Contact( "Unit1.EmNodes".allBrakeTest.monitoring.emStatus.busy[10] )
      I_Contact( "Unit1.EmNodes".allBrakeTest.monitoring.emStatus.busy[12] )
      I_Contact( "Unit1.EmNodes".allBrakeTest.monitoring.emStatus.busy[13] )
      I_Contact( "Unit1.EmNodes".allBrakeTest.monitoring.emStatus.busy[14] )
      I_Contact( "Unit1.EmNodes".allBrakeTest.monitoring.emStatus.busy[24] )
      I_Contact( "Unit1.EmNodes".allBrakeTest.monitoring.emStatus.busy[26] )
      I_Contact( "Unit1.EmNodes".allBrakeTest.monitoring.emStatus.busy[28] )
      I_Contact( "Unit1.EmNodes".allBrakeTest.monitoring.emStatus.busy[30] )
      I_Contact( "Unit1.EmNodes".allBrakeTest.monitoring.emStatus.busy[31] )
      I_Contact( "Unit1.EmNodes".allBrakeTest.monitoring.emStatus.busy[32] )
      I_Contact( "Unit1.EmNodes".allBrakeTest.monitoring.emStatus.busy[33] )
      I_Contact( "Unit1.EmNodes".allBrakeTest.monitoring.emStatus.busy[35] )
      I_Contact( "Unit1.EmNodes".allBrakeTest.monitoring.emStatus.busy[37] )
      Not()
      Coil( "Unit1.EmNodes".allBrakeTest.monitoring.allBusy )
      { S7_Templates := "time_type := Time" } #instTofTimer[8].TOF(pt := t#500ms, et =>)
      Coil( "Safety.DataToSafety".BrakeTest.allBrakeTesting )
   END_RUNG
   RUNG wire#powerrail
      Contact( "Unit1.EmNodes".allBrakeTest.monitoring.emStatus.complete[1] )
      Contact( "Unit1.EmNodes".allBrakeTest.monitoring.emStatus.complete[2] )
      Contact( "Unit1.EmNodes".allBrakeTest.monitoring.emStatus.complete[4] )
      Contact( "Unit1.EmNodes".allBrakeTest.monitoring.emStatus.complete[10] )
      Contact( "Unit1.EmNodes".allBrakeTest.monitoring.emStatus.complete[12] )
      Contact( "Unit1.EmNodes".allBrakeTest.monitoring.emStatus.complete[13] )
      Contact( "Unit1.EmNodes".allBrakeTest.monitoring.emStatus.complete[14] )
      Contact( "Unit1.EmNodes".allBrakeTest.monitoring.emStatus.complete[24] )
      Contact( "Unit1.EmNodes".allBrakeTest.monitoring.emStatus.complete[26] )
      Contact( "Unit1.EmNodes".allBrakeTest.monitoring.emStatus.complete[28] )
      Contact( "Unit1.EmNodes".allBrakeTest.monitoring.emStatus.complete[30] )
      Contact( "Unit1.EmNodes".allBrakeTest.monitoring.emStatus.complete[31] )
      Contact( "Unit1.EmNodes".allBrakeTest.monitoring.emStatus.complete[32] )
      Contact( "Unit1.EmNodes".allBrakeTest.monitoring.emStatus.complete[33] )
      Contact( "Unit1.EmNodes".allBrakeTest.monitoring.emStatus.complete[35] )
      Contact( "Unit1.EmNodes".allBrakeTest.monitoring.emStatus.complete[37] )
      wire#w1
      S_Coil( "Unit1.EmNodes".allBrakeTest.monitoring.firstScan )
   END_RUNG
   RUNG wire#w1
      Coil( "Unit1.EmNodes".allBrakeTest.monitoring.allComplete )
      Coil( "Safety.DataToSafety".BrakeTest.allBrakeTestDone )
   END_RUNG
   // the same network as SCL:
   "Unit1.EmNodes".allBrakeTest.monitoring.allBusy := NOT (NOT "Unit1.EmNodes".allBrakeTest.monitoring.emStatus.busy[1] AND NOT "Unit1.EmNodes".allBrakeTest.monitoring.emStatus.busy[2] AND NOT "Unit1.EmNodes".allBrakeTest.monitoring.emStatus.busy[4] AND NOT "Unit1.EmNodes".allBrakeTest.monitoring.emStatus.busy[10] AND NOT "Unit1.EmNodes".allBrakeTest.monitoring.emStatus.busy[12] AND NOT "Unit1.EmNodes".allBrakeTest.monitoring.emStatus.busy[13] AND NOT "Unit1.EmNodes".allBrakeTest.monitoring.emStatus.busy[14] AND NOT "Unit1.EmNodes".allBrakeTest.monitoring.emStatus.busy[24] AND NOT "Unit1.EmNodes".allBrakeTest.monitoring.emStatus.busy[26] AND NOT "Unit1.EmNodes".allBrakeTest.monitoring.emStatus.busy[28] AND NOT "Unit1.EmNodes".allBrakeTest.monitoring.emStatus.busy[30] AND NOT "Unit1.EmNodes".allBrakeTest.monitoring.emStatus.busy[31] AND NOT "Unit1.EmNodes".allBrakeTest.monitoring.emStatus.busy[32] AND NOT "Unit1.EmNodes".allBrakeTest.monitoring.emStatus.busy[33] AND NOT "Unit1.EmNodes".allBrakeTest.monitoring.emStatus.busy[35] AND NOT "Unit1.EmNodes".allBrakeTest.monitoring.emStatus.busy[37]);
   #instTofTimer[8].TOF(IN := "Unit1.EmNodes".allBrakeTest.monitoring.allBusy, PT := t#500ms);
   "Safety.DataToSafety".BrakeTest.allBrakeTesting := #instTofTimer[8].Q;
   #_w1 := "Unit1.EmNodes".allBrakeTest.monitoring.emStatus.complete[1] AND "Unit1.EmNodes".allBrakeTest.monitoring.emStatus.complete[2] AND "Unit1.EmNodes".allBrakeTest.monitoring.emStatus.complete[4] AND "Unit1.EmNodes".allBrakeTest.monitoring.emStatus.complete[10] AND "Unit1.EmNodes".allBrakeTest.monitoring.emStatus.complete[12] AND "Unit1.EmNodes".allBrakeTest.monitoring.emStatus.complete[13] AND "Unit1.EmNodes".allBrakeTest.monitoring.emStatus.complete[14] AND "Unit1.EmNodes".allBrakeTest.monitoring.emStatus.complete[24] AND "Unit1.EmNodes".allBrakeTest.monitoring.emStatus.complete[26] AND "Unit1.EmNodes".allBrakeTest.monitoring.emStatus.complete[28] AND "Unit1.EmNodes".allBrakeTest.monitoring.emStatus.complete[30] AND "Unit1.EmNodes".allBrakeTest.monitoring.emStatus.complete[31] AND "Unit1.EmNodes".allBrakeTest.monitoring.emStatus.complete[32] AND "Unit1.EmNodes".allBrakeTest.monitoring.emStatus.complete[33] AND "Unit1.EmNodes".allBrakeTest.monitoring.emStatus.complete[35] AND "Unit1.EmNodes".allBrakeTest.monitoring.emStatus.complete[37];
   IF #_w1 THEN "Unit1.EmNodes".allBrakeTest.monitoring.firstScan := TRUE; END_IF;
   "Unit1.EmNodes".allBrakeTest.monitoring.allComplete := #_w1;
   "Safety.DataToSafety".BrakeTest.allBrakeTestDone := #_w1;
END_REGION

REGION Network 86: Brake Test Time Check
   RUNG wire#powerrail
      Contact( "Unit1.EmNodes".allBrakeTest.monitoring.firstScan )
      I_Contact( "Unit1.EmNodes".allBrakeTest.monitoring.allComplete )
      wire#w1
      { S7_Templates := "time_type := Time" } #statTonTime[20].TON(pt := T#8h, et =>)
      I_Contact( "Unit1.EmNodes".allBrakeTest.monitoring.after24Hours )
      Coil( "Unit1.EmNodes".allBrakeTest.monitoring.after8Hours )
   END_RUNG
   RUNG wire#w1
      { S7_Templates := "time_type := Time" } #statTonTime[21].TON(pt := T#24h, et =>)
      Coil( "Unit1.EmNodes".allBrakeTest.monitoring.after24Hours )
   END_RUNG
   // the same network as SCL:
   #_w1 := "Unit1.EmNodes".allBrakeTest.monitoring.firstScan AND NOT "Unit1.EmNodes".allBrakeTest.monitoring.allComplete;
   #statTonTime[20].TON(IN := #_w1, PT := T#8h);
   "Unit1.EmNodes".allBrakeTest.monitoring.after8Hours := #statTonTime[20].Q AND NOT "Unit1.EmNodes".allBrakeTest.monitoring.after24Hours;
   #statTonTime[21].TON(IN := #_w1, PT := T#24h);
   "Unit1.EmNodes".allBrakeTest.monitoring.after24Hours := #statTonTime[21].Q;
END_REGION

REGION Network 87: All Brake Test Monitoring
   RUNG wire#powerrail
      Move(in := "Unit1.EmNodes".allBrakeTest.monitoring, out1 => "Unit1.HmiInterface".allBrakeTest.monitoring)
   END_RUNG
   // the same network as SCL:
   "Unit1.HmiInterface".allBrakeTest.monitoring := "Unit1.EmNodes".allBrakeTest.monitoring;
END_REGION

REGION Network 88: ******************** Motion Communication ********************
END_REGION

REGION Network 89: Stack Main Motion Ready
END_REGION

REGION Network 90: PLC To Motion Commands Stack Main Semi Step
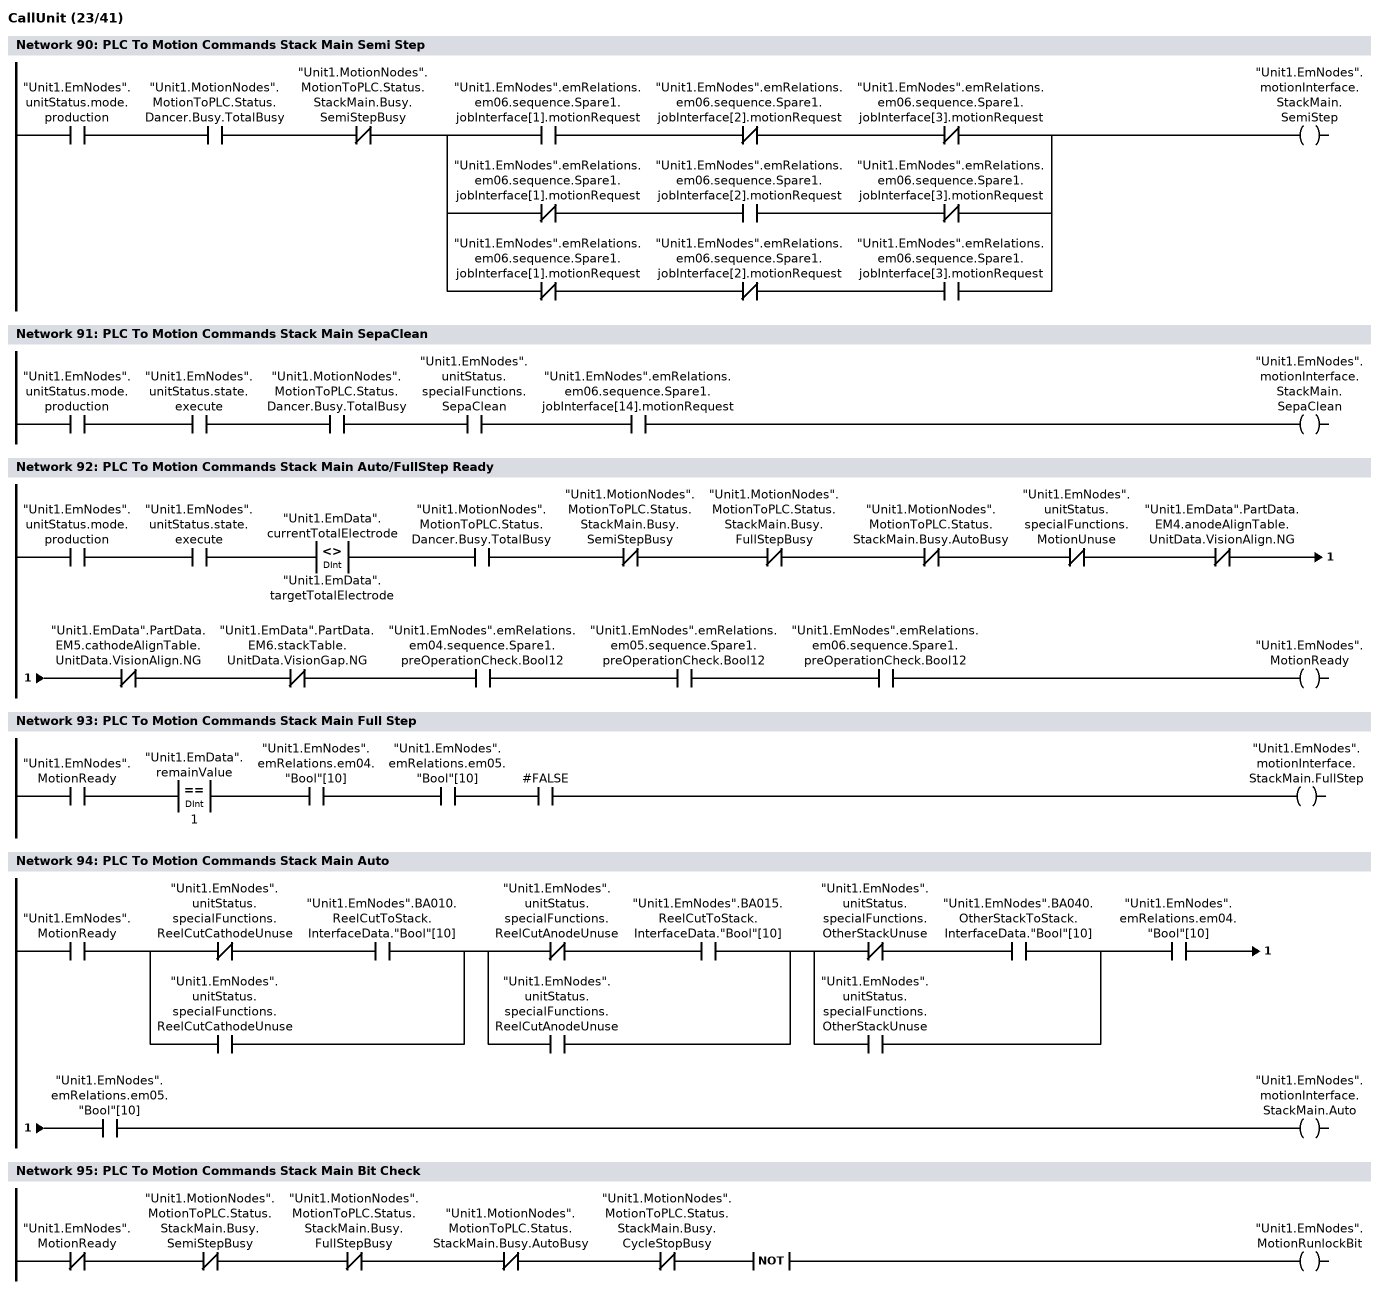
   RUNG wire#powerrail
      Contact( "Unit1.EmNodes".unitStatus.mode.production )
      Contact( "Unit1.MotionNodes".MotionToPLC.Status.Dancer.Busy.TotalBusy )
      I_Contact( "Unit1.MotionNodes".MotionToPLC.Status.StackMain.Busy.SemiStepBusy )
      wire#w1
      Contact( "Unit1.EmNodes".emRelations.em06.sequence.Spare1.jobInterface[1].motionRequest )
      I_Contact( "Unit1.EmNodes".emRelations.em06.sequence.Spare1.jobInterface[2].motionRequest )
      I_Contact( "Unit1.EmNodes".emRelations.em06.sequence.Spare1.jobInterface[3].motionRequest )
      wire#w2
      Coil( "Unit1.EmNodes".motionInterface.StackMain.SemiStep )
   END_RUNG
   RUNG wire#w1
      I_Contact( "Unit1.EmNodes".emRelations.em06.sequence.Spare1.jobInterface[1].motionRequest )
      Contact( "Unit1.EmNodes".emRelations.em06.sequence.Spare1.jobInterface[2].motionRequest )
      I_Contact( "Unit1.EmNodes".emRelations.em06.sequence.Spare1.jobInterface[3].motionRequest )
   END_RUNG wire#w2
   RUNG wire#w1
      I_Contact( "Unit1.EmNodes".emRelations.em06.sequence.Spare1.jobInterface[1].motionRequest )
      I_Contact( "Unit1.EmNodes".emRelations.em06.sequence.Spare1.jobInterface[2].motionRequest )
      Contact( "Unit1.EmNodes".emRelations.em06.sequence.Spare1.jobInterface[3].motionRequest )
   END_RUNG wire#w2
   // the same network as SCL:
   "Unit1.EmNodes".motionInterface.StackMain.SemiStep := "Unit1.EmNodes".unitStatus.mode.production AND "Unit1.MotionNodes".MotionToPLC.Status.Dancer.Busy.TotalBusy AND NOT "Unit1.MotionNodes".MotionToPLC.Status.StackMain.Busy.SemiStepBusy AND (("Unit1.EmNodes".emRelations.em06.sequence.Spare1.jobInterface[1].motionRequest AND NOT "Unit1.EmNodes".emRelations.em06.sequence.Spare1.jobInterface[2].motionRequest AND NOT "Unit1.EmNodes".emRelations.em06.sequence.Spare1.jobInterface[3].motionRequest) OR (NOT "Unit1.EmNodes".emRelations.em06.sequence.Spare1.jobInterface[1].motionRequest AND "Unit1.EmNodes".emRelations.em06.sequence.Spare1.jobInterface[2].motionRequest AND NOT "Unit1.EmNodes".emRelations.em06.sequence.Spare1.jobInterface[3].motionRequest) OR (NOT "Unit1.EmNodes".emRelations.em06.sequence.Spare1.jobInterface[1].motionRequest AND NOT "Unit1.EmNodes".emRelations.em06.sequence.Spare1.jobInterface[2].motionRequest AND "Unit1.EmNodes".emRelations.em06.sequence.Spare1.jobInterface[3].motionRequest));
END_REGION

REGION Network 91: PLC To Motion Commands Stack Main SepaClean
   RUNG wire#powerrail
      Contact( "Unit1.EmNodes".unitStatus.mode.production )
      Contact( "Unit1.EmNodes".unitStatus.state.execute )
      Contact( "Unit1.MotionNodes".MotionToPLC.Status.Dancer.Busy.TotalBusy )
      Contact( "Unit1.EmNodes".unitStatus.specialFunctions.SepaClean )
      Contact( "Unit1.EmNodes".emRelations.em06.sequence.Spare1.jobInterface[14].motionRequest )
      Coil( "Unit1.EmNodes".motionInterface.StackMain.SepaClean )
   END_RUNG
   // the same network as SCL:
   "Unit1.EmNodes".motionInterface.StackMain.SepaClean := "Unit1.EmNodes".unitStatus.mode.production AND "Unit1.EmNodes".unitStatus.state.execute AND "Unit1.MotionNodes".MotionToPLC.Status.Dancer.Busy.TotalBusy AND "Unit1.EmNodes".unitStatus.specialFunctions.SepaClean AND "Unit1.EmNodes".emRelations.em06.sequence.Spare1.jobInterface[14].motionRequest;
END_REGION

REGION Network 92: PLC To Motion Commands Stack Main Auto/FullStep Ready
   RUNG wire#powerrail
      Contact( "Unit1.EmNodes".unitStatus.mode.production )
      Contact( "Unit1.EmNodes".unitStatus.state.execute )
      { S7_Templates := "SrcType := DInt" } NE_Contact(in1 := "Unit1.EmData".currentTotalElectrode, in2 := "Unit1.EmData".targetTotalElectrode)
      Contact( "Unit1.MotionNodes".MotionToPLC.Status.Dancer.Busy.TotalBusy )
      I_Contact( "Unit1.MotionNodes".MotionToPLC.Status.StackMain.Busy.SemiStepBusy )
      I_Contact( "Unit1.MotionNodes".MotionToPLC.Status.StackMain.Busy.FullStepBusy )
      I_Contact( "Unit1.MotionNodes".MotionToPLC.Status.StackMain.Busy.AutoBusy )
      I_Contact( "Unit1.EmNodes".unitStatus.specialFunctions.MotionUnuse )
      I_Contact( "Unit1.EmData".PartData.EM4.anodeAlignTable.UnitData.VisionAlign.NG )
      I_Contact( "Unit1.EmData".PartData.EM5.cathodeAlignTable.UnitData.VisionAlign.NG )
      I_Contact( "Unit1.EmData".PartData.EM6.stackTable.UnitData.VisionGap.NG )
      Contact( "Unit1.EmNodes".emRelations.em04.sequence.Spare1.preOperationCheck.Bool12 )
      Contact( "Unit1.EmNodes".emRelations.em05.sequence.Spare1.preOperationCheck.Bool12 )
      Contact( "Unit1.EmNodes".emRelations.em06.sequence.Spare1.preOperationCheck.Bool12 )
      Coil( "Unit1.EmNodes".MotionReady )
   END_RUNG
   // the same network as SCL:
   "Unit1.EmNodes".MotionReady := "Unit1.EmNodes".unitStatus.mode.production AND "Unit1.EmNodes".unitStatus.state.execute AND ("Unit1.EmData".currentTotalElectrode <> "Unit1.EmData".targetTotalElectrode) AND "Unit1.MotionNodes".MotionToPLC.Status.Dancer.Busy.TotalBusy AND NOT "Unit1.MotionNodes".MotionToPLC.Status.StackMain.Busy.SemiStepBusy AND NOT "Unit1.MotionNodes".MotionToPLC.Status.StackMain.Busy.FullStepBusy AND NOT "Unit1.MotionNodes".MotionToPLC.Status.StackMain.Busy.AutoBusy AND NOT "Unit1.EmNodes".unitStatus.specialFunctions.MotionUnuse AND NOT "Unit1.EmData".PartData.EM4.anodeAlignTable.UnitData.VisionAlign.NG AND NOT "Unit1.EmData".PartData.EM5.cathodeAlignTable.UnitData.VisionAlign.NG AND NOT "Unit1.EmData".PartData.EM6.stackTable.UnitData.VisionGap.NG AND "Unit1.EmNodes".emRelations.em04.sequence.Spare1.preOperationCheck.Bool12 AND "Unit1.EmNodes".emRelations.em05.sequence.Spare1.preOperationCheck.Bool12 AND "Unit1.EmNodes".emRelations.em06.sequence.Spare1.preOperationCheck.Bool12;
END_REGION

REGION Network 93: PLC To Motion Commands Stack Main Full Step
   RUNG wire#powerrail
      Contact( "Unit1.EmNodes".MotionReady )
      { S7_Templates := "SrcType := DInt" } EQ_Contact(in1 := "Unit1.EmData".remainValue, in2 := 1)
      Contact( "Unit1.EmNodes".emRelations.em04."Bool"[10] )
      Contact( "Unit1.EmNodes".emRelations.em05."Bool"[10] )
      Contact( #FALSE )
      Coil( "Unit1.EmNodes".motionInterface.StackMain.FullStep )
   END_RUNG
   // the same network as SCL:
   "Unit1.EmNodes".motionInterface.StackMain.FullStep := "Unit1.EmNodes".MotionReady AND ("Unit1.EmData".remainValue = 1) AND "Unit1.EmNodes".emRelations.em04."Bool"[10] AND "Unit1.EmNodes".emRelations.em05."Bool"[10] AND #FALSE;
END_REGION

REGION Network 94: PLC To Motion Commands Stack Main Auto
   RUNG wire#powerrail
      Contact( "Unit1.EmNodes".MotionReady )
      wire#w1
      I_Contact( "Unit1.EmNodes".unitStatus.specialFunctions.ReelCutCathodeUnuse )
      Contact( "Unit1.EmNodes".BA010.ReelCutToStack.InterfaceData."Bool"[10] )
      wire#w2
      I_Contact( "Unit1.EmNodes".unitStatus.specialFunctions.ReelCutAnodeUnuse )
      Contact( "Unit1.EmNodes".BA015.ReelCutToStack.InterfaceData."Bool"[10] )
      wire#w3
      I_Contact( "Unit1.EmNodes".unitStatus.specialFunctions.OtherStackUnuse )
      Contact( "Unit1.EmNodes".BA040.OtherStackToStack.InterfaceData."Bool"[10] )
      wire#w4
      Contact( "Unit1.EmNodes".emRelations.em04."Bool"[10] )
      Contact( "Unit1.EmNodes".emRelations.em05."Bool"[10] )
      Coil( "Unit1.EmNodes".motionInterface.StackMain.Auto )
   END_RUNG
   RUNG wire#w1
      Contact( "Unit1.EmNodes".unitStatus.specialFunctions.ReelCutCathodeUnuse )
   END_RUNG wire#w2
   RUNG wire#w2
      Contact( "Unit1.EmNodes".unitStatus.specialFunctions.ReelCutAnodeUnuse )
   END_RUNG wire#w3
   RUNG wire#w3
      Contact( "Unit1.EmNodes".unitStatus.specialFunctions.OtherStackUnuse )
   END_RUNG wire#w4
   // the same network as SCL:
   "Unit1.EmNodes".motionInterface.StackMain.Auto := "Unit1.EmNodes".MotionReady AND ((NOT "Unit1.EmNodes".unitStatus.specialFunctions.ReelCutCathodeUnuse AND "Unit1.EmNodes".BA010.ReelCutToStack.InterfaceData."Bool"[10]) OR "Unit1.EmNodes".unitStatus.specialFunctions.ReelCutCathodeUnuse) AND ((NOT "Unit1.EmNodes".unitStatus.specialFunctions.ReelCutAnodeUnuse AND "Unit1.EmNodes".BA015.ReelCutToStack.InterfaceData."Bool"[10]) OR "Unit1.EmNodes".unitStatus.specialFunctions.ReelCutAnodeUnuse) AND ((NOT "Unit1.EmNodes".unitStatus.specialFunctions.OtherStackUnuse AND "Unit1.EmNodes".BA040.OtherStackToStack.InterfaceData."Bool"[10]) OR "Unit1.EmNodes".unitStatus.specialFunctions.OtherStackUnuse) AND "Unit1.EmNodes".emRelations.em04."Bool"[10] AND "Unit1.EmNodes".emRelations.em05."Bool"[10];
END_REGION

REGION Network 95: PLC To Motion Commands Stack Main Bit Check
   RUNG wire#powerrail
      I_Contact( "Unit1.EmNodes".MotionReady )
      I_Contact( "Unit1.MotionNodes".MotionToPLC.Status.StackMain.Busy.SemiStepBusy )
      I_Contact( "Unit1.MotionNodes".MotionToPLC.Status.StackMain.Busy.FullStepBusy )
      I_Contact( "Unit1.MotionNodes".MotionToPLC.Status.StackMain.Busy.AutoBusy )
      I_Contact( "Unit1.MotionNodes".MotionToPLC.Status.StackMain.Busy.CycleStopBusy )
      Not()
      Coil( "Unit1.EmNodes".MotionRunlockBit )
   END_RUNG
   // the same network as SCL:
   "Unit1.EmNodes".MotionRunlockBit := NOT (NOT "Unit1.EmNodes".MotionReady AND NOT "Unit1.MotionNodes".MotionToPLC.Status.StackMain.Busy.SemiStepBusy AND NOT "Unit1.MotionNodes".MotionToPLC.Status.StackMain.Busy.FullStepBusy AND NOT "Unit1.MotionNodes".MotionToPLC.Status.StackMain.Busy.AutoBusy AND NOT "Unit1.MotionNodes".MotionToPLC.Status.StackMain.Busy.CycleStopBusy);
END_REGION

REGION Network 96: PLC To Motion Commands Stack Main Stop
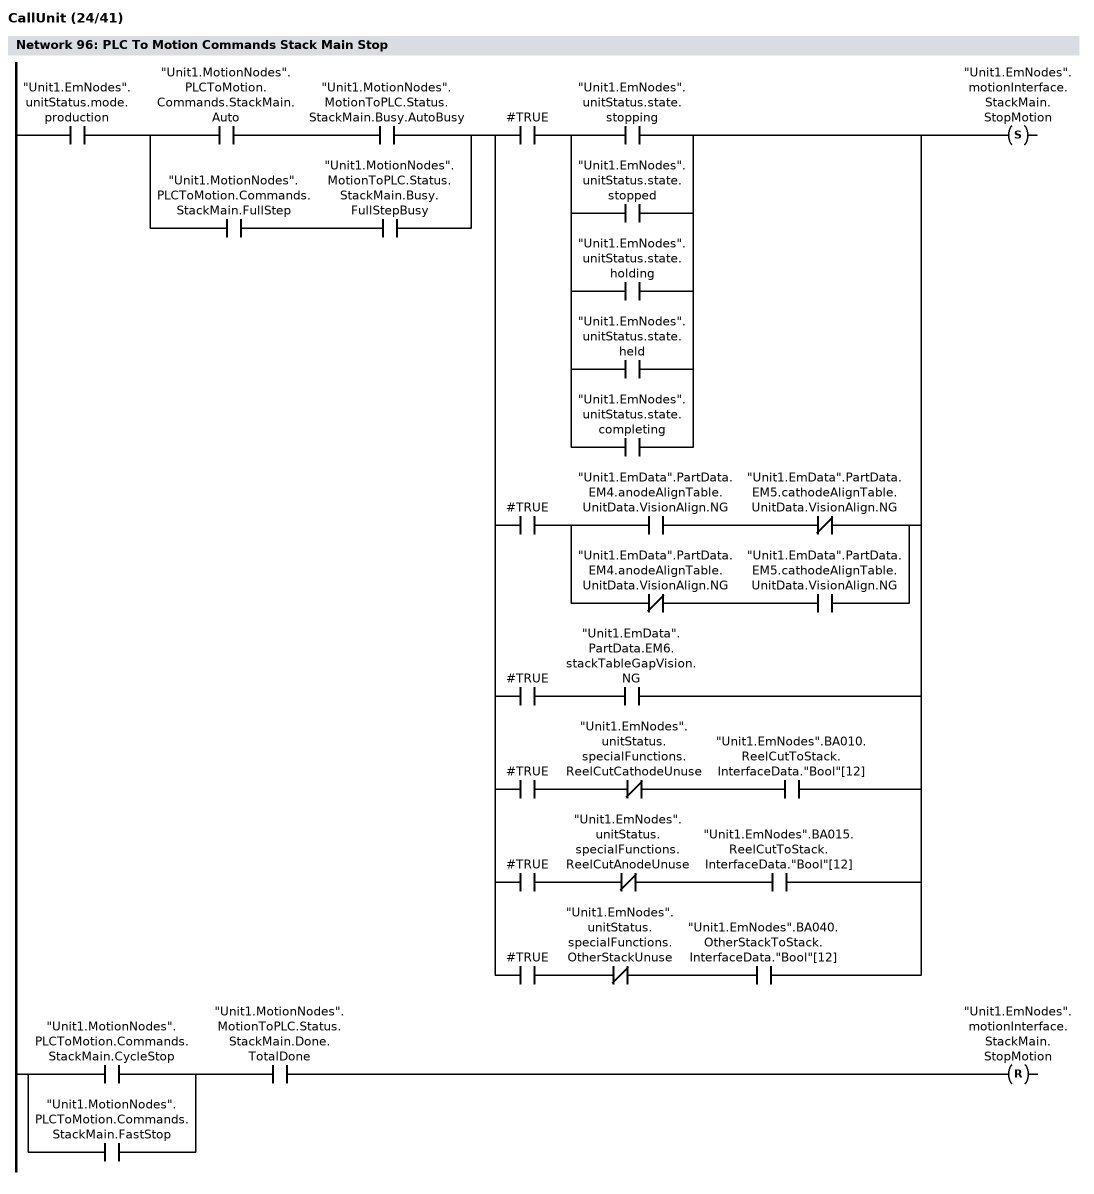
   RUNG wire#powerrail
      Contact( "Unit1.EmNodes".unitStatus.mode.production )
      wire#w1
      Contact( "Unit1.MotionNodes".PLCToMotion.Commands.StackMain.Auto )
      Contact( "Unit1.MotionNodes".MotionToPLC.Status.StackMain.Busy.AutoBusy )
      wire#w2
      Contact( #TRUE )
      wire#w3
      Contact( "Unit1.EmNodes".unitStatus.state.stopping )
      wire#w4
      S_Coil( "Unit1.EmNodes".motionInterface.StackMain.StopMotion )
   END_RUNG
   RUNG wire#w1
      Contact( "Unit1.MotionNodes".PLCToMotion.Commands.StackMain.FullStep )
      Contact( "Unit1.MotionNodes".MotionToPLC.Status.StackMain.Busy.FullStepBusy )
   END_RUNG wire#w2
   RUNG wire#w3
      Contact( "Unit1.EmNodes".unitStatus.state.stopped )
   END_RUNG wire#w4
   RUNG wire#w3
      Contact( "Unit1.EmNodes".unitStatus.state.holding )
   END_RUNG wire#w4
   RUNG wire#w3
      Contact( "Unit1.EmNodes".unitStatus.state.held )
   END_RUNG wire#w4
   RUNG wire#w3
      Contact( "Unit1.EmNodes".unitStatus.state.completing )
   END_RUNG wire#w4
   RUNG wire#w2
      Contact( #TRUE )
      wire#w5
      Contact( "Unit1.EmData".PartData.EM4.anodeAlignTable.UnitData.VisionAlign.NG )
      I_Contact( "Unit1.EmData".PartData.EM5.cathodeAlignTable.UnitData.VisionAlign.NG )
   END_RUNG wire#w4
   RUNG wire#w5
      I_Contact( "Unit1.EmData".PartData.EM4.anodeAlignTable.UnitData.VisionAlign.NG )
      Contact( "Unit1.EmData".PartData.EM5.cathodeAlignTable.UnitData.VisionAlign.NG )
   END_RUNG wire#w4
   RUNG wire#w2
      Contact( #TRUE )
      Contact( "Unit1.EmData".PartData.EM6.stackTableGapVision.NG )
   END_RUNG wire#w4
   RUNG wire#w2
      Contact( #TRUE )
      I_Contact( "Unit1.EmNodes".unitStatus.specialFunctions.ReelCutCathodeUnuse )
      Contact( "Unit1.EmNodes".BA010.ReelCutToStack.InterfaceData."Bool"[12] )
   END_RUNG wire#w4
   RUNG wire#w2
      Contact( #TRUE )
      I_Contact( "Unit1.EmNodes".unitStatus.specialFunctions.ReelCutAnodeUnuse )
      Contact( "Unit1.EmNodes".BA015.ReelCutToStack.InterfaceData."Bool"[12] )
   END_RUNG wire#w4
   RUNG wire#w2
      Contact( #TRUE )
      I_Contact( "Unit1.EmNodes".unitStatus.specialFunctions.OtherStackUnuse )
      Contact( "Unit1.EmNodes".BA040.OtherStackToStack.InterfaceData."Bool"[12] )
   END_RUNG wire#w4
   RUNG wire#powerrail
      Contact( "Unit1.MotionNodes".PLCToMotion.Commands.StackMain.CycleStop )
      wire#w6
      Contact( "Unit1.MotionNodes".MotionToPLC.Status.StackMain.Done.TotalDone )
      R_Coil( "Unit1.EmNodes".motionInterface.StackMain.StopMotion )
   END_RUNG
   RUNG wire#powerrail
      Contact( "Unit1.MotionNodes".PLCToMotion.Commands.StackMain.FastStop )
   END_RUNG wire#w6
   // the same network as SCL:
   IF "Unit1.EmNodes".unitStatus.mode.production AND (("Unit1.MotionNodes".PLCToMotion.Commands.StackMain.Auto AND "Unit1.MotionNodes".MotionToPLC.Status.StackMain.Busy.AutoBusy) OR ("Unit1.MotionNodes".PLCToMotion.Commands.StackMain.FullStep AND "Unit1.MotionNodes".MotionToPLC.Status.StackMain.Busy.FullStepBusy)) AND ((#TRUE AND ("Unit1.EmNodes".unitStatus.state.stopping OR "Unit1.EmNodes".unitStatus.state.stopped OR "Unit1.EmNodes".unitStatus.state.holding OR "Unit1.EmNodes".unitStatus.state.held OR "Unit1.EmNodes".unitStatus.state.completing)) OR (#TRUE AND (("Unit1.EmData".PartData.EM4.anodeAlignTable.UnitData.VisionAlign.NG AND NOT "Unit1.EmData".PartData.EM5.cathodeAlignTable.UnitData.VisionAlign.NG) OR (NOT "Unit1.EmData".PartData.EM4.anodeAlignTable.UnitData.VisionAlign.NG AND "Unit1.EmData".PartData.EM5.cathodeAlignTable.UnitData.VisionAlign.NG))) OR (#TRUE AND "Unit1.EmData".PartData.EM6.stackTableGapVision.NG) OR (#TRUE AND NOT "Unit1.EmNodes".unitStatus.specialFunctions.ReelCutCathodeUnuse AND "Unit1.EmNodes".BA010.ReelCutToStack.InterfaceData."Bool"[12]) OR (#TRUE AND NOT "Unit1.EmNodes".unitStatus.specialFunctions.ReelCutAnodeUnuse AND "Unit1.EmNodes".BA015.ReelCutToStack.InterfaceData."Bool"[12]) OR (#TRUE AND NOT "Unit1.EmNodes".unitStatus.specialFunctions.OtherStackUnuse AND "Unit1.EmNodes".BA040.OtherStackToStack.InterfaceData."Bool"[12])) THEN
       "Unit1.EmNodes".motionInterface.StackMain.StopMotion := TRUE;
   END_IF;
   IF ("Unit1.MotionNodes".PLCToMotion.Commands.StackMain.CycleStop OR "Unit1.MotionNodes".PLCToMotion.Commands.StackMain.FastStop) AND "Unit1.MotionNodes".MotionToPLC.Status.StackMain.Done.TotalDone THEN
       "Unit1.EmNodes".motionInterface.StackMain.StopMotion := FALSE;
   END_IF;
END_REGION

REGION Network 97: PLC To Motion Commands Stack Main
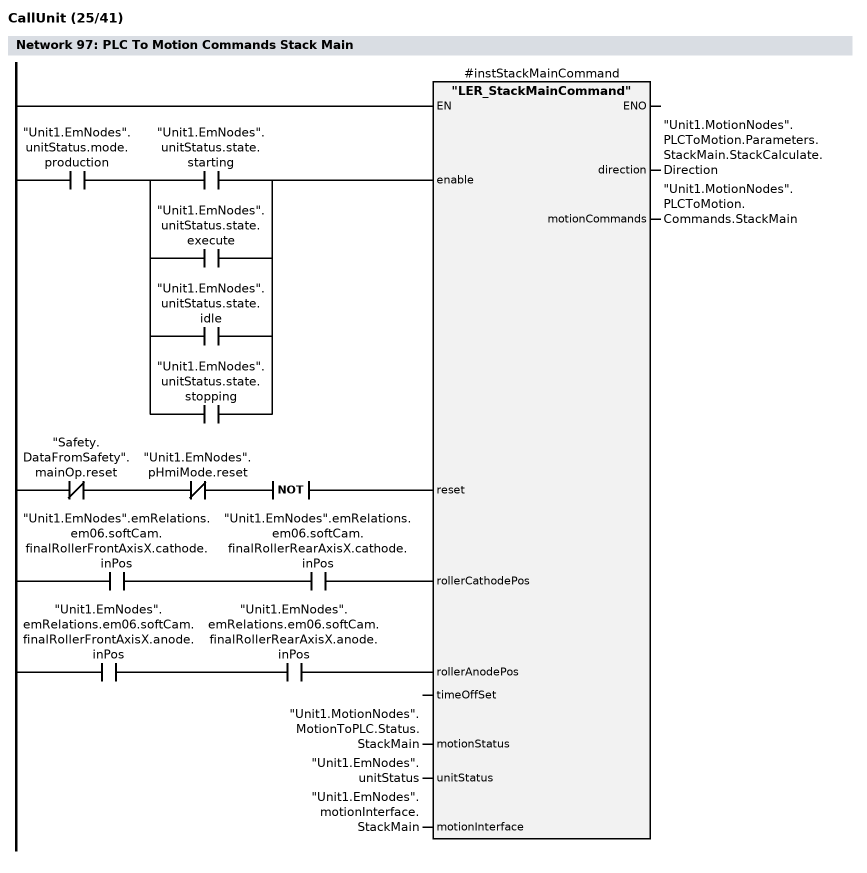
   RUNG wire#powerrail
      #instStackMainCommand(enable := wire#w2, reset := wire#w3, rollerCathodePos := wire#w4, rollerAnodePos := wire#w5, timeOffSet :=, motionStatus := "Unit1.MotionNodes".MotionToPLC.Status.StackMain, unitStatus := "Unit1.EmNodes".unitStatus, motionInterface := "Unit1.EmNodes".motionInterface.StackMain, direction => "Unit1.MotionNodes".PLCToMotion.Parameters.StackMain.StackCalculate.Direction, motionCommands => "Unit1.MotionNodes".PLCToMotion.Commands.StackMain)
   END_RUNG
   RUNG wire#powerrail
      Contact( "Unit1.EmNodes".unitStatus.mode.production )
      wire#w1
      Contact( "Unit1.EmNodes".unitStatus.state.starting )
   END_RUNG wire#w2
   RUNG wire#w1
      Contact( "Unit1.EmNodes".unitStatus.state.execute )
   END_RUNG wire#w2
   RUNG wire#w1
      Contact( "Unit1.EmNodes".unitStatus.state.idle )
   END_RUNG wire#w2
   RUNG wire#w1
      Contact( "Unit1.EmNodes".unitStatus.state.stopping )
   END_RUNG wire#w2
   RUNG wire#powerrail
      I_Contact( "Safety.DataFromSafety".mainOp.reset )
      I_Contact( "Unit1.EmNodes".pHmiMode.reset )
      Not()
   END_RUNG wire#w3
   RUNG wire#powerrail
      Contact( "Unit1.EmNodes".emRelations.em06.softCam.finalRollerFrontAxisX.cathode.inPos )
      Contact( "Unit1.EmNodes".emRelations.em06.softCam.finalRollerRearAxisX.cathode.inPos )
   END_RUNG wire#w4
   RUNG wire#powerrail
      Contact( "Unit1.EmNodes".emRelations.em06.softCam.finalRollerFrontAxisX.anode.inPos )
      Contact( "Unit1.EmNodes".emRelations.em06.softCam.finalRollerRearAxisX.anode.inPos )
   END_RUNG wire#w5
   // the same network as SCL:
   #instStackMainCommand(enable := "Unit1.EmNodes".unitStatus.mode.production AND ("Unit1.EmNodes".unitStatus.state.starting OR "Unit1.EmNodes".unitStatus.state.execute OR "Unit1.EmNodes".unitStatus.state.idle OR "Unit1.EmNodes".unitStatus.state.stopping),   // "LER_StackMainCommand"
                         reset := NOT (NOT "Safety.DataFromSafety".mainOp.reset AND NOT "Unit1.EmNodes".pHmiMode.reset),
                         rollerCathodePos := "Unit1.EmNodes".emRelations.em06.softCam.finalRollerFrontAxisX.cathode.inPos AND "Unit1.EmNodes".emRelations.em06.softCam.finalRollerRearAxisX.cathode.inPos,
                         rollerAnodePos := "Unit1.EmNodes".emRelations.em06.softCam.finalRollerFrontAxisX.anode.inPos AND "Unit1.EmNodes".emRelations.em06.softCam.finalRollerRearAxisX.anode.inPos,
                         motionStatus := "Unit1.MotionNodes".MotionToPLC.Status.StackMain,
                         unitStatus := "Unit1.EmNodes".unitStatus,
                         motionInterface := "Unit1.EmNodes".motionInterface.StackMain,
                         direction => "Unit1.MotionNodes".PLCToMotion.Parameters.StackMain.StackCalculate.Direction,
                         motionCommands => "Unit1.MotionNodes".PLCToMotion.Commands.StackMain);
END_REGION

REGION Network 98: PLC To Motion Commands Dancer
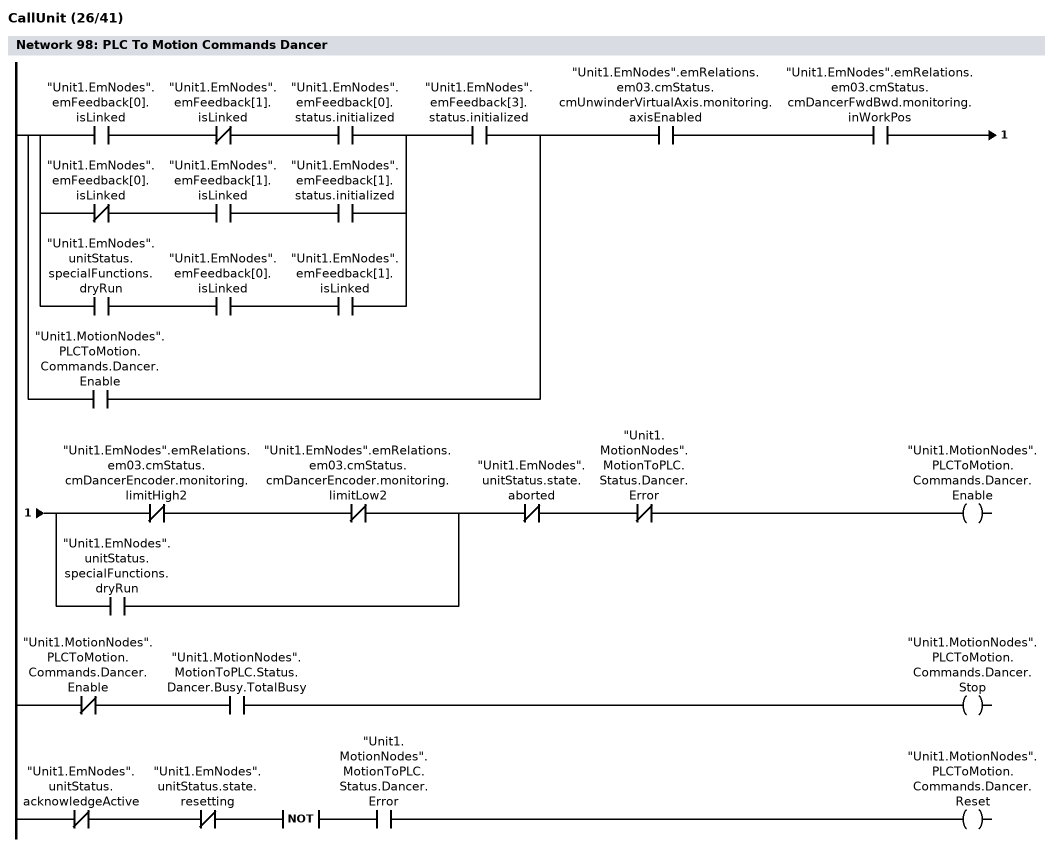
   RUNG wire#powerrail
      Contact( "Unit1.EmNodes".emFeedback[0].isLinked )
      I_Contact( "Unit1.EmNodes".emFeedback[1].isLinked )
      Contact( "Unit1.EmNodes".emFeedback[0].status.initialized )
      wire#w1
      Contact( "Unit1.EmNodes".emFeedback[3].status.initialized )
      wire#w2
      Contact( "Unit1.EmNodes".emRelations.em03.cmStatus.cmUnwinderVirtualAxis.monitoring.axisEnabled )
      Contact( "Unit1.EmNodes".emRelations.em03.cmStatus.cmDancerFwdBwd.monitoring.inWorkPos )
      wire#w3
      I_Contact( "Unit1.EmNodes".emRelations.em03.cmStatus.cmDancerEncoder.monitoring.limitHigh2 )
      I_Contact( "Unit1.EmNodes".emRelations.em03.cmStatus.cmDancerEncoder.monitoring.limitLow2 )
      wire#w4
      I_Contact( "Unit1.EmNodes".unitStatus.state.aborted )
      I_Contact( "Unit1.MotionNodes".MotionToPLC.Status.Dancer.Error )
      Coil( "Unit1.MotionNodes".PLCToMotion.Commands.Dancer.Enable )
   END_RUNG
   RUNG wire#powerrail
      I_Contact( "Unit1.EmNodes".emFeedback[0].isLinked )
      Contact( "Unit1.EmNodes".emFeedback[1].isLinked )
      Contact( "Unit1.EmNodes".emFeedback[1].status.initialized )
   END_RUNG wire#w1
   RUNG wire#powerrail
      Contact( "Unit1.EmNodes".unitStatus.specialFunctions.dryRun )
      Contact( "Unit1.EmNodes".emFeedback[0].isLinked )
      Contact( "Unit1.EmNodes".emFeedback[1].isLinked )
   END_RUNG wire#w1
   RUNG wire#powerrail
      Contact( "Unit1.MotionNodes".PLCToMotion.Commands.Dancer.Enable )
   END_RUNG wire#w2
   RUNG wire#w3
      Contact( "Unit1.EmNodes".unitStatus.specialFunctions.dryRun )
   END_RUNG wire#w4
   RUNG wire#powerrail
      I_Contact( "Unit1.MotionNodes".PLCToMotion.Commands.Dancer.Enable )
      Contact( "Unit1.MotionNodes".MotionToPLC.Status.Dancer.Busy.TotalBusy )
      Coil( "Unit1.MotionNodes".PLCToMotion.Commands.Dancer.Stop )
   END_RUNG
   RUNG wire#powerrail
      I_Contact( "Unit1.EmNodes".unitStatus.acknowledgeActive )
      I_Contact( "Unit1.EmNodes".unitStatus.state.resetting )
      Not()
      Contact( "Unit1.MotionNodes".MotionToPLC.Status.Dancer.Error )
      Coil( "Unit1.MotionNodes".PLCToMotion.Commands.Dancer.Reset )
   END_RUNG
   // the same network as SCL:
   "Unit1.MotionNodes".PLCToMotion.Commands.Dancer.Enable := (((("Unit1.EmNodes".emFeedback[0].isLinked AND NOT "Unit1.EmNodes".emFeedback[1].isLinked AND "Unit1.EmNodes".emFeedback[0].status.initialized) OR (NOT "Unit1.EmNodes".emFeedback[0].isLinked AND "Unit1.EmNodes".emFeedback[1].isLinked AND "Unit1.EmNodes".emFeedback[1].status.initialized) OR ("Unit1.EmNodes".unitStatus.specialFunctions.dryRun AND "Unit1.EmNodes".emFeedback[0].isLinked AND "Unit1.EmNodes".emFeedback[1].isLinked)) AND "Unit1.EmNodes".emFeedback[3].status.initialized) OR "Unit1.MotionNodes".PLCToMotion.Commands.Dancer.Enable) AND "Unit1.EmNodes".emRelations.em03.cmStatus.cmUnwinderVirtualAxis.monitoring.axisEnabled AND "Unit1.EmNodes".emRelations.em03.cmStatus.cmDancerFwdBwd.monitoring.inWorkPos AND ((NOT "Unit1.EmNodes".emRelations.em03.cmStatus.cmDancerEncoder.monitoring.limitHigh2 AND NOT "Unit1.EmNodes".emRelations.em03.cmStatus.cmDancerEncoder.monitoring.limitLow2) OR "Unit1.EmNodes".unitStatus.specialFunctions.dryRun) AND NOT "Unit1.EmNodes".unitStatus.state.aborted AND NOT "Unit1.MotionNodes".MotionToPLC.Status.Dancer.Error;
   "Unit1.MotionNodes".PLCToMotion.Commands.Dancer.Stop := NOT "Unit1.MotionNodes".PLCToMotion.Commands.Dancer.Enable AND "Unit1.MotionNodes".MotionToPLC.Status.Dancer.Busy.TotalBusy;
   "Unit1.MotionNodes".PLCToMotion.Commands.Dancer.Reset := NOT (NOT "Unit1.EmNodes".unitStatus.acknowledgeActive AND NOT "Unit1.EmNodes".unitStatus.state.resetting) AND "Unit1.MotionNodes".MotionToPLC.Status.Dancer.Error;
END_REGION

REGION Network 99: PLC To Motion InitialPos Mapping
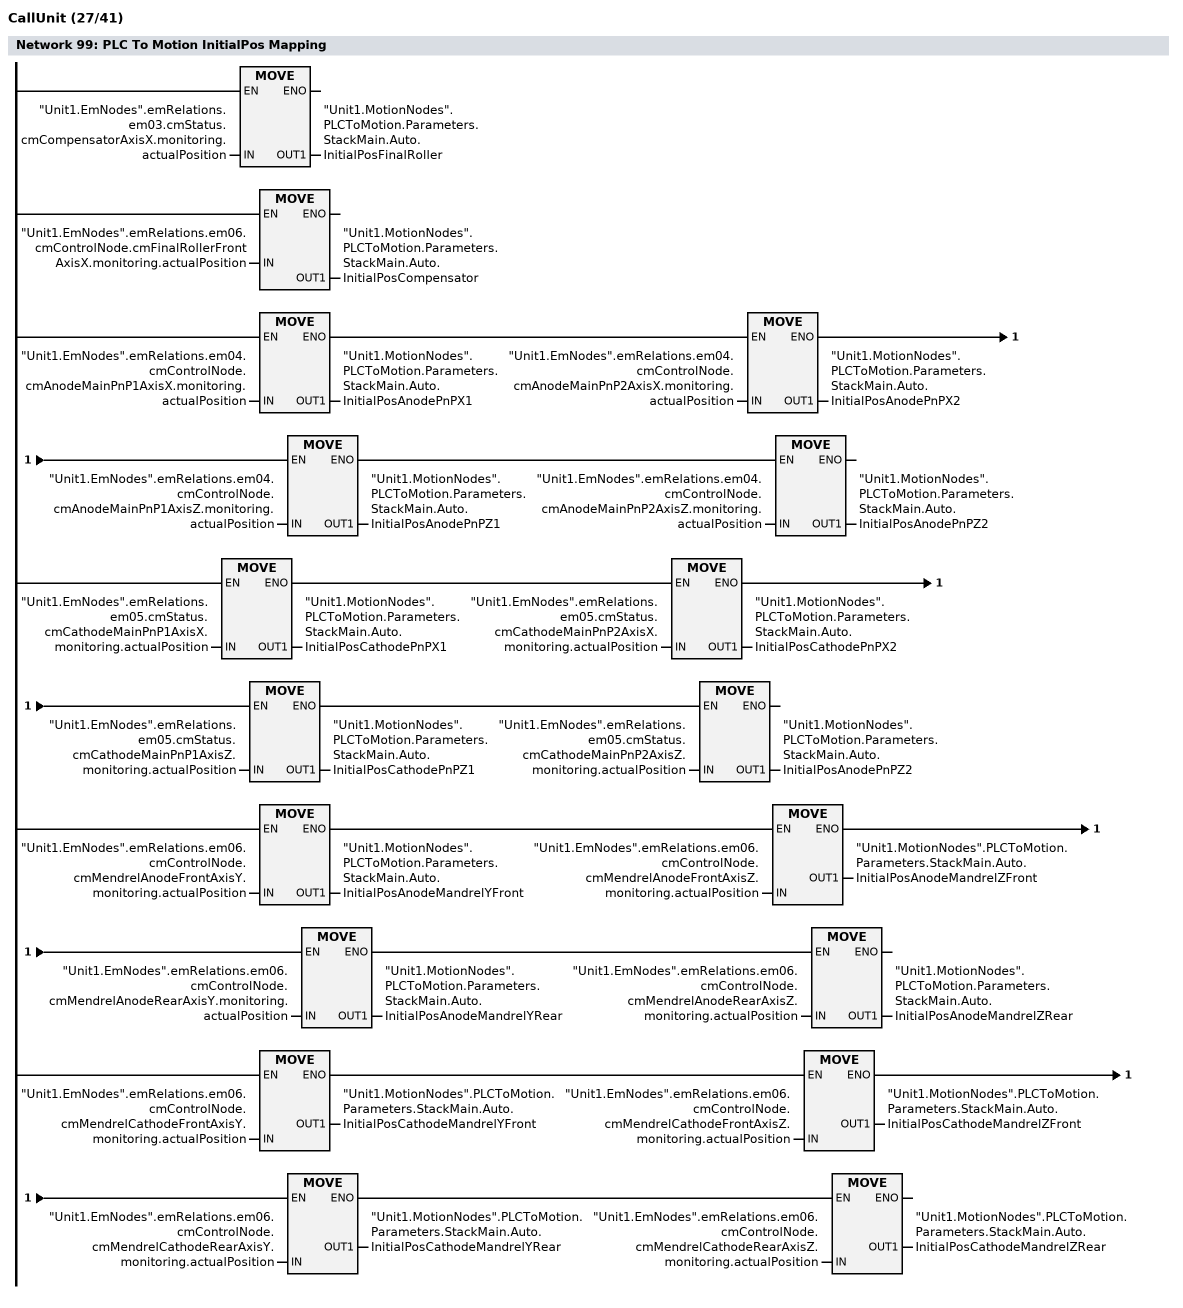
   RUNG wire#powerrail
      Move(in := "Unit1.EmNodes".emRelations.em03.cmStatus.cmCompensatorAxisX.monitoring.actualPosition, out1 => "Unit1.MotionNodes".PLCToMotion.Parameters.StackMain.Auto.InitialPosFinalRoller)
   END_RUNG
   RUNG wire#powerrail
      Move(in := "Unit1.EmNodes".emRelations.em06.cmControlNode.cmFinalRollerFrontAxisX.monitoring.actualPosition, out1 => "Unit1.MotionNodes".PLCToMotion.Parameters.StackMain.Auto.InitialPosCompensator)
   END_RUNG
   RUNG wire#powerrail
      Move(in := "Unit1.EmNodes".emRelations.em04.cmControlNode.cmAnodeMainPnP1AxisX.monitoring.actualPosition, out1 => "Unit1.MotionNodes".PLCToMotion.Parameters.StackMain.Auto.InitialPosAnodePnPX1)
      Move(in := "Unit1.EmNodes".emRelations.em04.cmControlNode.cmAnodeMainPnP2AxisX.monitoring.actualPosition, out1 => "Unit1.MotionNodes".PLCToMotion.Parameters.StackMain.Auto.InitialPosAnodePnPX2)
      Move(in := "Unit1.EmNodes".emRelations.em04.cmControlNode.cmAnodeMainPnP1AxisZ.monitoring.actualPosition, out1 => "Unit1.MotionNodes".PLCToMotion.Parameters.StackMain.Auto.InitialPosAnodePnPZ1)
      Move(in := "Unit1.EmNodes".emRelations.em04.cmControlNode.cmAnodeMainPnP2AxisZ.monitoring.actualPosition, out1 => "Unit1.MotionNodes".PLCToMotion.Parameters.StackMain.Auto.InitialPosAnodePnPZ2)
   END_RUNG
   RUNG wire#powerrail
      Move(in := "Unit1.EmNodes".emRelations.em05.cmStatus.cmCathodeMainPnP1AxisX.monitoring.actualPosition, out1 => "Unit1.MotionNodes".PLCToMotion.Parameters.StackMain.Auto.InitialPosCathodePnPX1)
      Move(in := "Unit1.EmNodes".emRelations.em05.cmStatus.cmCathodeMainPnP2AxisX.monitoring.actualPosition, out1 => "Unit1.MotionNodes".PLCToMotion.Parameters.StackMain.Auto.InitialPosCathodePnPX2)
      Move(in := "Unit1.EmNodes".emRelations.em05.cmStatus.cmCathodeMainPnP1AxisZ.monitoring.actualPosition, out1 => "Unit1.MotionNodes".PLCToMotion.Parameters.StackMain.Auto.InitialPosCathodePnPZ1)
      Move(in := "Unit1.EmNodes".emRelations.em05.cmStatus.cmCathodeMainPnP2AxisZ.monitoring.actualPosition, out1 => "Unit1.MotionNodes".PLCToMotion.Parameters.StackMain.Auto.InitialPosAnodePnPZ2)
   END_RUNG
   RUNG wire#powerrail
      Move(in := "Unit1.EmNodes".emRelations.em06.cmControlNode.cmMendrelAnodeFrontAxisY.monitoring.actualPosition, out1 => "Unit1.MotionNodes".PLCToMotion.Parameters.StackMain.Auto.InitialPosAnodeMandrelYFront)
      Move(in := "Unit1.EmNodes".emRelations.em06.cmControlNode.cmMendrelAnodeFrontAxisZ.monitoring.actualPosition, out1 => "Unit1.MotionNodes".PLCToMotion.Parameters.StackMain.Auto.InitialPosAnodeMandrelZFront)
      Move(in := "Unit1.EmNodes".emRelations.em06.cmControlNode.cmMendrelAnodeRearAxisY.monitoring.actualPosition, out1 => "Unit1.MotionNodes".PLCToMotion.Parameters.StackMain.Auto.InitialPosAnodeMandrelYRear)
      Move(in := "Unit1.EmNodes".emRelations.em06.cmControlNode.cmMendrelAnodeRearAxisZ.monitoring.actualPosition, out1 => "Unit1.MotionNodes".PLCToMotion.Parameters.StackMain.Auto.InitialPosAnodeMandrelZRear)
   END_RUNG
   RUNG wire#powerrail
      Move(in := "Unit1.EmNodes".emRelations.em06.cmControlNode.cmMendrelCathodeFrontAxisY.monitoring.actualPosition, out1 => "Unit1.MotionNodes".PLCToMotion.Parameters.StackMain.Auto.InitialPosCathodeMandrelYFront)
      Move(in := "Unit1.EmNodes".emRelations.em06.cmControlNode.cmMendrelCathodeFrontAxisZ.monitoring.actualPosition, out1 => "Unit1.MotionNodes".PLCToMotion.Parameters.StackMain.Auto.InitialPosCathodeMandrelZFront)
      Move(in := "Unit1.EmNodes".emRelations.em06.cmControlNode.cmMendrelCathodeRearAxisY.monitoring.actualPosition, out1 => "Unit1.MotionNodes".PLCToMotion.Parameters.StackMain.Auto.InitialPosCathodeMandrelYRear)
      Move(in := "Unit1.EmNodes".emRelations.em06.cmControlNode.cmMendrelCathodeRearAxisZ.monitoring.actualPosition, out1 => "Unit1.MotionNodes".PLCToMotion.Parameters.StackMain.Auto.InitialPosCathodeMandrelZRear)
   END_RUNG
   // the same network as SCL:
   "Unit1.MotionNodes".PLCToMotion.Parameters.StackMain.Auto.InitialPosFinalRoller := "Unit1.EmNodes".emRelations.em03.cmStatus.cmCompensatorAxisX.monitoring.actualPosition;
   "Unit1.MotionNodes".PLCToMotion.Parameters.StackMain.Auto.InitialPosCompensator := "Unit1.EmNodes".emRelations.em06.cmControlNode.cmFinalRollerFrontAxisX.monitoring.actualPosition;
   "Unit1.MotionNodes".PLCToMotion.Parameters.StackMain.Auto.InitialPosAnodePnPX1 := "Unit1.EmNodes".emRelations.em04.cmControlNode.cmAnodeMainPnP1AxisX.monitoring.actualPosition;
   "Unit1.MotionNodes".PLCToMotion.Parameters.StackMain.Auto.InitialPosAnodePnPX2 := "Unit1.EmNodes".emRelations.em04.cmControlNode.cmAnodeMainPnP2AxisX.monitoring.actualPosition;
   "Unit1.MotionNodes".PLCToMotion.Parameters.StackMain.Auto.InitialPosAnodePnPZ1 := "Unit1.EmNodes".emRelations.em04.cmControlNode.cmAnodeMainPnP1AxisZ.monitoring.actualPosition;
   "Unit1.MotionNodes".PLCToMotion.Parameters.StackMain.Auto.InitialPosAnodePnPZ2 := "Unit1.EmNodes".emRelations.em04.cmControlNode.cmAnodeMainPnP2AxisZ.monitoring.actualPosition;
   "Unit1.MotionNodes".PLCToMotion.Parameters.StackMain.Auto.InitialPosCathodePnPX1 := "Unit1.EmNodes".emRelations.em05.cmStatus.cmCathodeMainPnP1AxisX.monitoring.actualPosition;
   "Unit1.MotionNodes".PLCToMotion.Parameters.StackMain.Auto.InitialPosCathodePnPX2 := "Unit1.EmNodes".emRelations.em05.cmStatus.cmCathodeMainPnP2AxisX.monitoring.actualPosition;
   "Unit1.MotionNodes".PLCToMotion.Parameters.StackMain.Auto.InitialPosCathodePnPZ1 := "Unit1.EmNodes".emRelations.em05.cmStatus.cmCathodeMainPnP1AxisZ.monitoring.actualPosition;
   "Unit1.MotionNodes".PLCToMotion.Parameters.StackMain.Auto.InitialPosAnodePnPZ2 := "Unit1.EmNodes".emRelations.em05.cmStatus.cmCathodeMainPnP2AxisZ.monitoring.actualPosition;
   "Unit1.MotionNodes".PLCToMotion.Parameters.StackMain.Auto.InitialPosAnodeMandrelYFront := "Unit1.EmNodes".emRelations.em06.cmControlNode.cmMendrelAnodeFrontAxisY.monitoring.actualPosition;
   "Unit1.MotionNodes".PLCToMotion.Parameters.StackMain.Auto.InitialPosAnodeMandrelZFront := "Unit1.EmNodes".emRelations.em06.cmControlNode.cmMendrelAnodeFrontAxisZ.monitoring.actualPosition;
   "Unit1.MotionNodes".PLCToMotion.Parameters.StackMain.Auto.InitialPosAnodeMandrelYRear := "Unit1.EmNodes".emRelations.em06.cmControlNode.cmMendrelAnodeRearAxisY.monitoring.actualPosition;
   "Unit1.MotionNodes".PLCToMotion.Parameters.StackMain.Auto.InitialPosAnodeMandrelZRear := "Unit1.EmNodes".emRelations.em06.cmControlNode.cmMendrelAnodeRearAxisZ.monitoring.actualPosition;
   "Unit1.MotionNodes".PLCToMotion.Parameters.StackMain.Auto.InitialPosCathodeMandrelYFront := "Unit1.EmNodes".emRelations.em06.cmControlNode.cmMendrelCathodeFrontAxisY.monitoring.actualPosition;
   "Unit1.MotionNodes".PLCToMotion.Parameters.StackMain.Auto.InitialPosCathodeMandrelZFront := "Unit1.EmNodes".emRelations.em06.cmControlNode.cmMendrelCathodeFrontAxisZ.monitoring.actualPosition;
   "Unit1.MotionNodes".PLCToMotion.Parameters.StackMain.Auto.InitialPosCathodeMandrelYRear := "Unit1.EmNodes".emRelations.em06.cmControlNode.cmMendrelCathodeRearAxisY.monitoring.actualPosition;
   "Unit1.MotionNodes".PLCToMotion.Parameters.StackMain.Auto.InitialPosCathodeMandrelZRear := "Unit1.EmNodes".emRelations.em06.cmControlNode.cmMendrelCathodeRearAxisZ.monitoring.actualPosition;
END_REGION

REGION Network 100: ******************** Calculate ********************
END_REGION

REGION Network 101: Currnet ToTal Electrode Number
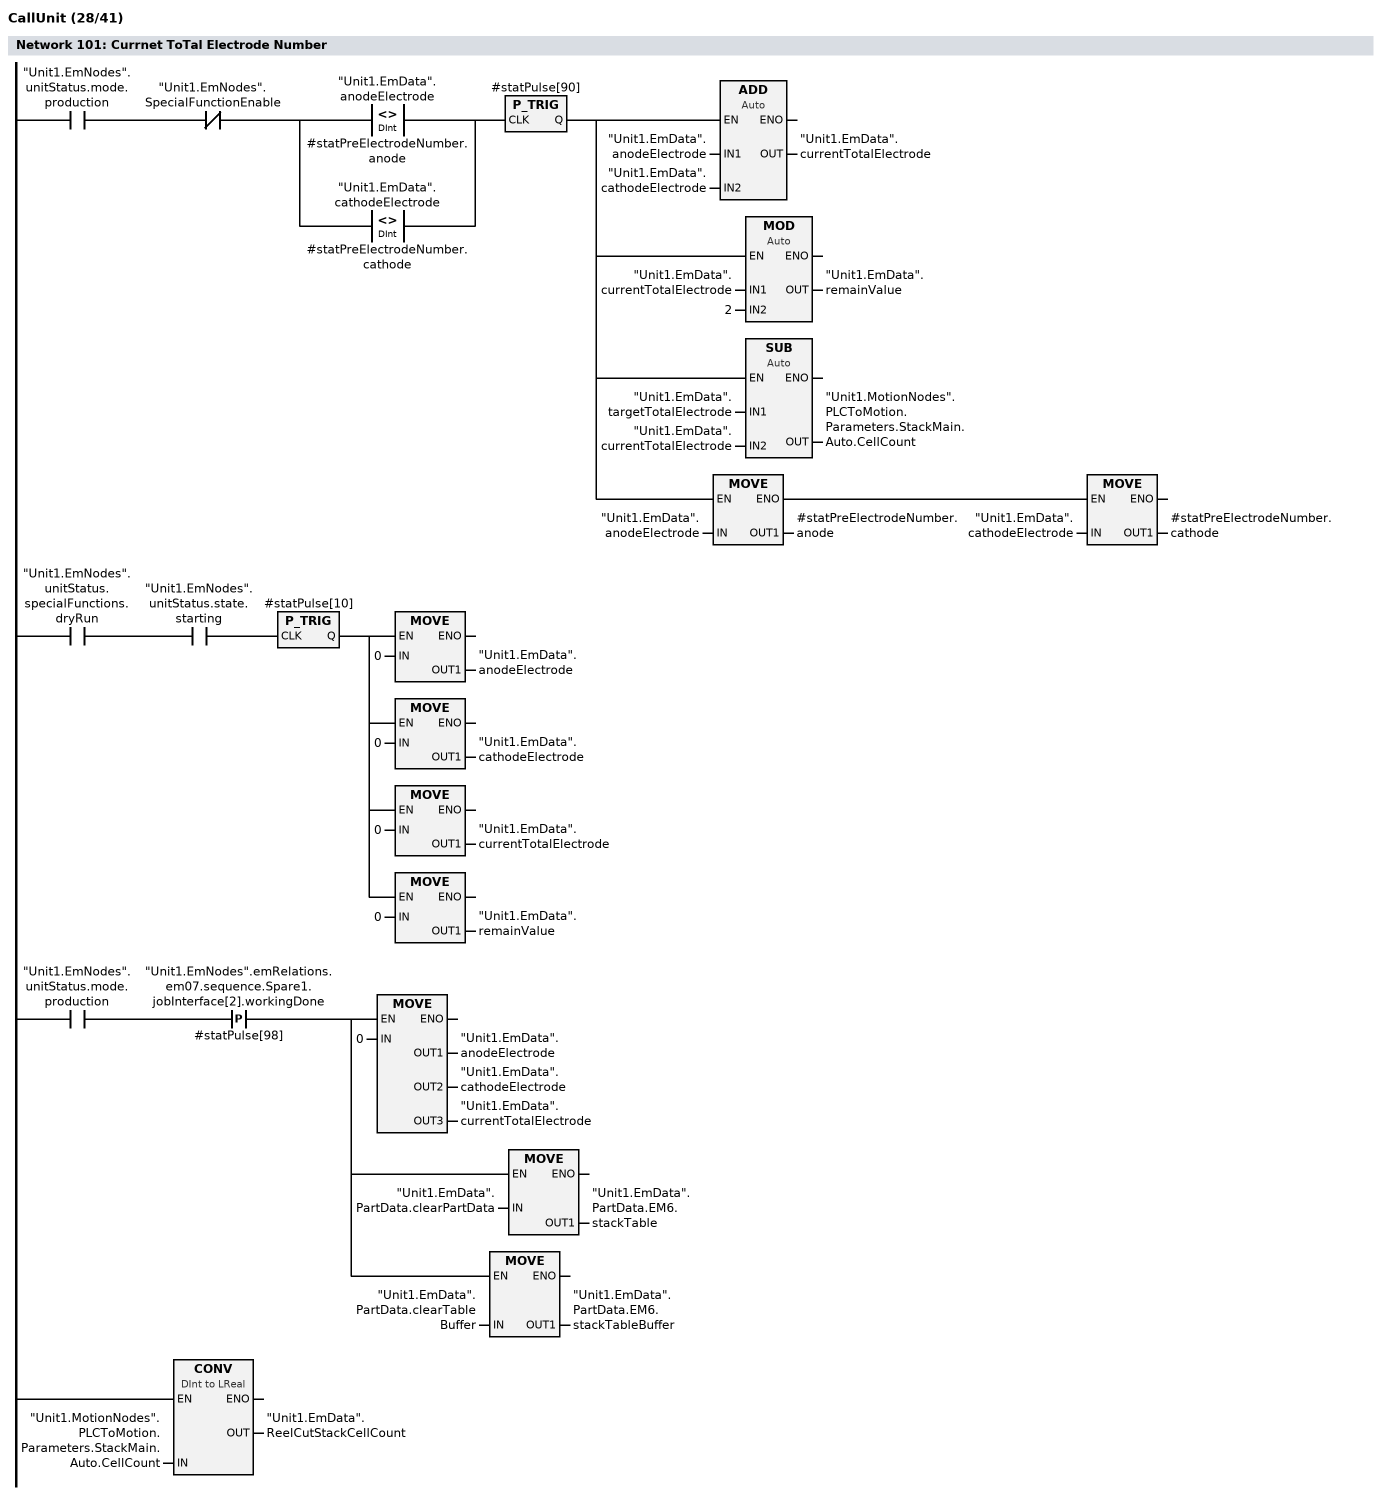
   RUNG wire#powerrail
      Contact( "Unit1.EmNodes".unitStatus.mode.production )
      I_Contact( "Unit1.EmNodes".SpecialFunctionEnable )
      wire#w1
      { S7_Templates := "SrcType := DInt" } NE_Contact(in1 := "Unit1.EmData".anodeElectrode, in2 := #statPreElectrodeNumber.anode)
      wire#w2
      P_Trig( #statPulse[90] )
      wire#w3
      Add(in1 := "Unit1.EmData".anodeElectrode, in2 := "Unit1.EmData".cathodeElectrode, out => "Unit1.EmData".currentTotalElectrode)
   END_RUNG
   RUNG wire#w1
      { S7_Templates := "SrcType := DInt" } NE_Contact(in1 := "Unit1.EmData".cathodeElectrode, in2 := #statPreElectrodeNumber.cathode)
   END_RUNG wire#w2
   RUNG wire#w3
      Mod(in1 := "Unit1.EmData".currentTotalElectrode, in2 := 2, out => "Unit1.EmData".remainValue)
   END_RUNG
   RUNG wire#w3
      Sub(in1 := "Unit1.EmData".targetTotalElectrode, in2 := "Unit1.EmData".currentTotalElectrode, out => "Unit1.MotionNodes".PLCToMotion.Parameters.StackMain.Auto.CellCount)
   END_RUNG
   RUNG wire#w3
      Move(in := "Unit1.EmData".anodeElectrode, out1 => #statPreElectrodeNumber.anode)
      Move(in := "Unit1.EmData".cathodeElectrode, out1 => #statPreElectrodeNumber.cathode)
   END_RUNG
   RUNG wire#powerrail
      Contact( "Unit1.EmNodes".unitStatus.specialFunctions.dryRun )
      Contact( "Unit1.EmNodes".unitStatus.state.starting )
      P_Trig( #statPulse[10] )
      wire#w4
      Move(in := 0, out1 => "Unit1.EmData".anodeElectrode)
   END_RUNG
   RUNG wire#w4
      Move(in := 0, out1 => "Unit1.EmData".cathodeElectrode)
   END_RUNG
   RUNG wire#w4
      Move(in := 0, out1 => "Unit1.EmData".currentTotalElectrode)
   END_RUNG
   RUNG wire#w4
      Move(in := 0, out1 => "Unit1.EmData".remainValue)
   END_RUNG
   RUNG wire#powerrail
      Contact( "Unit1.EmNodes".unitStatus.mode.production )
      P_Contact(operand := "Unit1.EmNodes".emRelations.em07.sequence.Spare1.jobInterface[2].workingDone, bit := #statPulse[98])
      wire#w5
      Move(in := 0, out1 => "Unit1.EmData".anodeElectrode, out2 => "Unit1.EmData".cathodeElectrode, out3 => "Unit1.EmData".currentTotalElectrode)
   END_RUNG
   RUNG wire#w5
      Move(in := "Unit1.EmData".PartData.clearPartData, out1 => "Unit1.EmData".PartData.EM6.stackTable)
   END_RUNG
   RUNG wire#w5
      Move(in := "Unit1.EmData".PartData.clearTableBuffer, out1 => "Unit1.EmData".PartData.EM6.stackTableBuffer)
   END_RUNG
   RUNG wire#powerrail
      { S7_Templates := "[SrcType := DInt, DestType := LReal]" } Convert(in := "Unit1.MotionNodes".PLCToMotion.Parameters.StackMain.Auto.CellCount, out => "Unit1.EmData".ReelCutStackCellCount)
   END_RUNG
   // the same network as SCL:
   #_w1 := "Unit1.EmNodes".unitStatus.mode.production AND NOT "Unit1.EmNodes".SpecialFunctionEnable AND (("Unit1.EmData".anodeElectrode <> #statPreElectrodeNumber.anode) OR ("Unit1.EmData".cathodeElectrode <> #statPreElectrodeNumber.cathode));
   #_w2 := #_w1 AND NOT #statPulse[90];   // rising edge
   #statPulse[90] := #_w1;
   IF #_w2 THEN
       "Unit1.EmData".currentTotalElectrode := "Unit1.EmData".anodeElectrode + "Unit1.EmData".cathodeElectrode;
       "Unit1.EmData".remainValue := "Unit1.EmData".currentTotalElectrode MOD 2;
       "Unit1.MotionNodes".PLCToMotion.Parameters.StackMain.Auto.CellCount := "Unit1.EmData".targetTotalElectrode - "Unit1.EmData".currentTotalElectrode;
       #statPreElectrodeNumber.anode := "Unit1.EmData".anodeElectrode;
       #statPreElectrodeNumber.cathode := "Unit1.EmData".cathodeElectrode;
   END_IF;
   #_w3 := "Unit1.EmNodes".unitStatus.specialFunctions.dryRun AND "Unit1.EmNodes".unitStatus.state.starting;
   #_w4 := #_w3 AND NOT #statPulse[10];   // rising edge
   #statPulse[10] := #_w3;
   IF #_w4 THEN
       "Unit1.EmData".anodeElectrode := 0;
       "Unit1.EmData".cathodeElectrode := 0;
       "Unit1.EmData".currentTotalElectrode := 0;
       "Unit1.EmData".remainValue := 0;
   END_IF;
   #_w5 := "Unit1.EmNodes".unitStatus.mode.production AND "Unit1.EmNodes".emRelations.em07.sequence.Spare1.jobInterface[2].workingDone AND NOT #statPulse[98];   // rising edge of "Unit1.EmNodes".emRelations.em07.sequence.Spare1.jobInterface[2].workingDone
   #statPulse[98] := "Unit1.EmNodes".emRelations.em07.sequence.Spare1.jobInterface[2].workingDone;
   IF #_w5 THEN
       "Unit1.EmData".anodeElectrode := 0;
       "Unit1.EmData".cathodeElectrode := 0;
       "Unit1.EmData".currentTotalElectrode := 0;
       "Unit1.EmData".PartData.EM6.stackTable := "Unit1.EmData".PartData.clearPartData;
       "Unit1.EmData".PartData.EM6.stackTableBuffer := "Unit1.EmData".PartData.clearTableBuffer;
   END_IF;
   "Unit1.EmData".ReelCutStackCellCount := DINT_TO_LREAL("Unit1.MotionNodes".PLCToMotion.Parameters.StackMain.Auto.CellCount);
END_REGION

REGION Network 102: Current Total Production Quantity
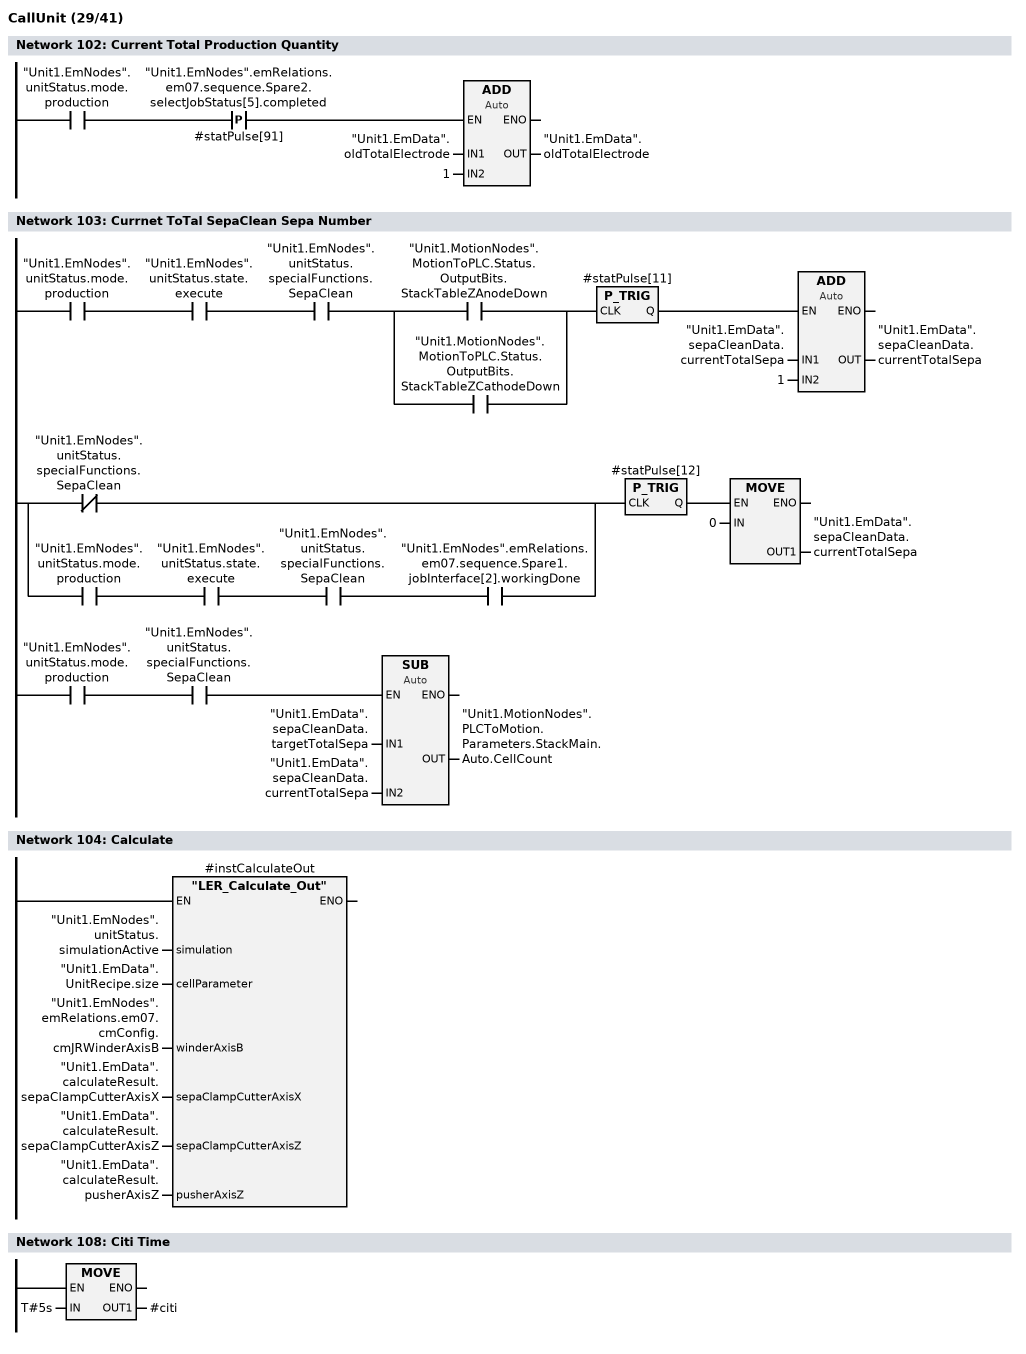
   RUNG wire#powerrail
      Contact( "Unit1.EmNodes".unitStatus.mode.production )
      P_Contact(operand := "Unit1.EmNodes".emRelations.em07.sequence.Spare2.selectJobStatus[5].completed, bit := #statPulse[91])
      Add(in1 := "Unit1.EmData".oldTotalElectrode, in2 := 1, out => "Unit1.EmData".oldTotalElectrode)
   END_RUNG
   // the same network as SCL:
   #_w1 := "Unit1.EmNodes".unitStatus.mode.production AND "Unit1.EmNodes".emRelations.em07.sequence.Spare2.selectJobStatus[5].completed AND NOT #statPulse[91];   // rising edge of "Unit1.EmNodes".emRelations.em07.sequence.Spare2.selectJobStatus[5].completed
   #statPulse[91] := "Unit1.EmNodes".emRelations.em07.sequence.Spare2.selectJobStatus[5].completed;
   IF #_w1 THEN "Unit1.EmData".oldTotalElectrode := "Unit1.EmData".oldTotalElectrode + 1; END_IF;
END_REGION

REGION Network 103: Currnet ToTal SepaClean Sepa Number
   RUNG wire#powerrail
      Contact( "Unit1.EmNodes".unitStatus.mode.production )
      Contact( "Unit1.EmNodes".unitStatus.state.execute )
      Contact( "Unit1.EmNodes".unitStatus.specialFunctions.SepaClean )
      wire#w1
      Contact( "Unit1.MotionNodes".MotionToPLC.Status.OutputBits.StackTableZAnodeDown )
      wire#w2
      P_Trig( #statPulse[11] )
      Add(in1 := "Unit1.EmData".sepaCleanData.currentTotalSepa, in2 := 1, out => "Unit1.EmData".sepaCleanData.currentTotalSepa)
   END_RUNG
   RUNG wire#w1
      Contact( "Unit1.MotionNodes".MotionToPLC.Status.OutputBits.StackTableZCathodeDown )
   END_RUNG wire#w2
   RUNG wire#powerrail
      I_Contact( "Unit1.EmNodes".unitStatus.specialFunctions.SepaClean )
      wire#w3
      P_Trig( #statPulse[12] )
      Move(in := 0, out1 => "Unit1.EmData".sepaCleanData.currentTotalSepa)
   END_RUNG
   RUNG wire#powerrail
      Contact( "Unit1.EmNodes".unitStatus.mode.production )
      Contact( "Unit1.EmNodes".unitStatus.state.execute )
      Contact( "Unit1.EmNodes".unitStatus.specialFunctions.SepaClean )
      Contact( "Unit1.EmNodes".emRelations.em07.sequence.Spare1.jobInterface[2].workingDone )
   END_RUNG wire#w3
   RUNG wire#powerrail
      Contact( "Unit1.EmNodes".unitStatus.mode.production )
      Contact( "Unit1.EmNodes".unitStatus.specialFunctions.SepaClean )
      Sub(in1 := "Unit1.EmData".sepaCleanData.targetTotalSepa, in2 := "Unit1.EmData".sepaCleanData.currentTotalSepa, out => "Unit1.MotionNodes".PLCToMotion.Parameters.StackMain.Auto.CellCount)
   END_RUNG
   // the same network as SCL:
   #_w1 := "Unit1.EmNodes".unitStatus.mode.production AND "Unit1.EmNodes".unitStatus.state.execute AND "Unit1.EmNodes".unitStatus.specialFunctions.SepaClean AND ("Unit1.MotionNodes".MotionToPLC.Status.OutputBits.StackTableZAnodeDown OR "Unit1.MotionNodes".MotionToPLC.Status.OutputBits.StackTableZCathodeDown);
   #_w2 := #_w1 AND NOT #statPulse[11];   // rising edge
   #statPulse[11] := #_w1;
   IF #_w2 THEN
       "Unit1.EmData".sepaCleanData.currentTotalSepa := "Unit1.EmData".sepaCleanData.currentTotalSepa + 1;
   END_IF;
   #_w3 := NOT "Unit1.EmNodes".unitStatus.specialFunctions.SepaClean OR ("Unit1.EmNodes".unitStatus.mode.production AND "Unit1.EmNodes".unitStatus.state.execute AND "Unit1.EmNodes".unitStatus.specialFunctions.SepaClean AND "Unit1.EmNodes".emRelations.em07.sequence.Spare1.jobInterface[2].workingDone);
   #_w4 := #_w3 AND NOT #statPulse[12];   // rising edge
   #statPulse[12] := #_w3;
   IF #_w4 THEN "Unit1.EmData".sepaCleanData.currentTotalSepa := 0; END_IF;
   IF "Unit1.EmNodes".unitStatus.mode.production AND "Unit1.EmNodes".unitStatus.specialFunctions.SepaClean THEN
       "Unit1.MotionNodes".PLCToMotion.Parameters.StackMain.Auto.CellCount := "Unit1.EmData".sepaCleanData.targetTotalSepa - "Unit1.EmData".sepaCleanData.currentTotalSepa;
   END_IF;
END_REGION

REGION Network 104: Calculate
   RUNG wire#powerrail
      #instCalculateOut(simulation := "Unit1.EmNodes".unitStatus.simulationActive, cellParameter := "Unit1.EmData".UnitRecipe.size, winderAxisB := "Unit1.EmNodes".emRelations.em07.cmConfig.cmJRWinderAxisB, sepaClampCutterAxisX := "Unit1.EmData".calculateResult.sepaClampCutterAxisX, sepaClampCutterAxisZ := "Unit1.EmData".calculateResult.sepaClampCutterAxisZ, pusherAxisZ := "Unit1.EmData".calculateResult.pusherAxisZ)
   END_RUNG
   // the same network as SCL:
   #instCalculateOut(simulation := "Unit1.EmNodes".unitStatus.simulationActive,   // "LER_Calculate_Out"
                     cellParameter := "Unit1.EmData".UnitRecipe.size,
                     winderAxisB := "Unit1.EmNodes".emRelations.em07.cmConfig.cmJRWinderAxisB,
                     sepaClampCutterAxisX := "Unit1.EmData".calculateResult.sepaClampCutterAxisX,
                     sepaClampCutterAxisZ := "Unit1.EmData".calculateResult.sepaClampCutterAxisZ,
                     pusherAxisZ := "Unit1.EmData".calculateResult.pusherAxisZ);
END_REGION

REGION Network 105 (SCL): Calculate Total Sepa Web Lenth
   #statCalculateParameters.AnodeCount := ("Unit1.EmData".targetTotalElectrode + 1) / 2;
   #statCalculateParameters.CathodeCount := ("Unit1.EmData".targetTotalElectrode - 1) / 2;
   #statCalculateParameters.SepaCount := "Unit1.EmData".targetTotalElectrode;

   #statCalculateParameters.TotalThickness := (#statCalculateParameters.AnodeCount * "Unit1.EmData".UnitRecipe.size.Anode.thickness) + (#statCalculateParameters.CathodeCount * "Unit1.EmData".UnitRecipe.size.Cathode.thickness) + (#statCalculateParameters.SepaCount * "Unit1.EmData".UnitRecipe.SepaThickness);

   "Unit1.EmData".UnitRecipe.TotalSepaWebLenth:= ("Unit1.EmData".UnitRecipe.JellyRollWidth * 3.5) + (#statCalculateParameters.TotalThickness * 3);
END_REGION

REGION Network 107: ******************** CITI ********************
END_REGION

REGION Network 108: Citi Time
   RUNG wire#powerrail
      Move(in := T#5s, out1 => #citi)
   END_RUNG
   // the same network as SCL:
   #citi := T#5s;
END_REGION

REGION Network 109: Auto Cycle Running 0
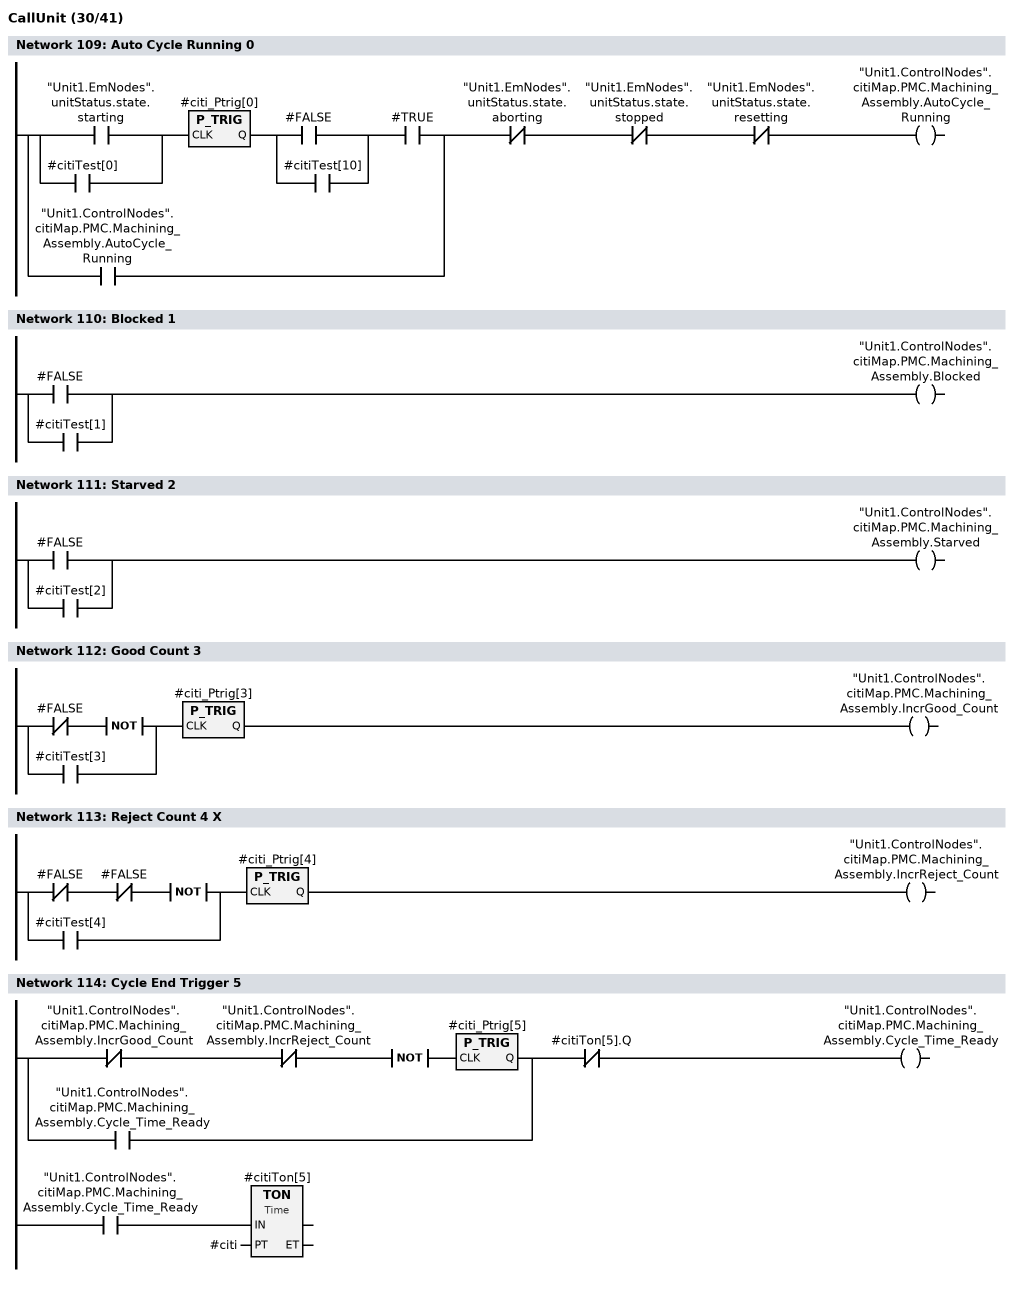
   RUNG wire#powerrail
      Contact( "Unit1.EmNodes".unitStatus.state.starting )
      wire#w1
      P_Trig( #citi_Ptrig[0] )
      wire#w2
      Contact( #FALSE )
      wire#w3
      Contact( #TRUE )
      wire#w4
      I_Contact( "Unit1.EmNodes".unitStatus.state.aborting )
      I_Contact( "Unit1.EmNodes".unitStatus.state.stopped )
      I_Contact( "Unit1.EmNodes".unitStatus.state.resetting )
      Coil( "Unit1.ControlNodes".citiMap.PMC.Machining_Assembly.AutoCycle_Running )
   END_RUNG
   RUNG wire#powerrail
      Contact( #citiTest[0] )
   END_RUNG wire#w1
   RUNG wire#w2
      Contact( #citiTest[10] )
   END_RUNG wire#w3
   RUNG wire#powerrail
      Contact( "Unit1.ControlNodes".citiMap.PMC.Machining_Assembly.AutoCycle_Running )
   END_RUNG wire#w4
   // the same network as SCL:
   #_w1 := "Unit1.EmNodes".unitStatus.state.starting OR #citiTest[0];
   #_w2 := #_w1 AND NOT #citi_Ptrig[0];   // rising edge
   #citi_Ptrig[0] := #_w1;
   "Unit1.ControlNodes".citiMap.PMC.Machining_Assembly.AutoCycle_Running := ((#_w2 AND (#FALSE OR #citiTest[10]) AND #TRUE) OR "Unit1.ControlNodes".citiMap.PMC.Machining_Assembly.AutoCycle_Running) AND NOT "Unit1.EmNodes".unitStatus.state.aborting AND NOT "Unit1.EmNodes".unitStatus.state.stopped AND NOT "Unit1.EmNodes".unitStatus.state.resetting;
END_REGION

REGION Network 110: Blocked 1
   RUNG wire#powerrail
      Contact( #FALSE )
      wire#w1
      Coil( "Unit1.ControlNodes".citiMap.PMC.Machining_Assembly.Blocked )
   END_RUNG
   RUNG wire#powerrail
      Contact( #citiTest[1] )
   END_RUNG wire#w1
   // the same network as SCL:
   "Unit1.ControlNodes".citiMap.PMC.Machining_Assembly.Blocked := #FALSE OR #citiTest[1];
END_REGION

REGION Network 111: Starved 2
   RUNG wire#powerrail
      Contact( #FALSE )
      wire#w1
      Coil( "Unit1.ControlNodes".citiMap.PMC.Machining_Assembly.Starved )
   END_RUNG
   RUNG wire#powerrail
      Contact( #citiTest[2] )
   END_RUNG wire#w1
   // the same network as SCL:
   "Unit1.ControlNodes".citiMap.PMC.Machining_Assembly.Starved := #FALSE OR #citiTest[2];
END_REGION

REGION Network 112: Good Count 3
   RUNG wire#powerrail
      I_Contact( #FALSE )
      Not()
      wire#w1
      P_Trig( #citi_Ptrig[3] )
      Coil( "Unit1.ControlNodes".citiMap.PMC.Machining_Assembly.IncrGood_Count )
   END_RUNG
   RUNG wire#powerrail
      Contact( #citiTest[3] )
   END_RUNG wire#w1
   // the same network as SCL:
   #_w1 := NOT (NOT #FALSE) OR #citiTest[3];
   #_w2 := #_w1 AND NOT #citi_Ptrig[3];   // rising edge
   #citi_Ptrig[3] := #_w1;
   "Unit1.ControlNodes".citiMap.PMC.Machining_Assembly.IncrGood_Count := #_w2;
END_REGION

REGION Network 113: Reject Count 4 X
   RUNG wire#powerrail
      I_Contact( #FALSE )
      I_Contact( #FALSE )
      Not()
      wire#w1
      P_Trig( #citi_Ptrig[4] )
      Coil( "Unit1.ControlNodes".citiMap.PMC.Machining_Assembly.IncrReject_Count )
   END_RUNG
   RUNG wire#powerrail
      Contact( #citiTest[4] )
   END_RUNG wire#w1
   // the same network as SCL:
   #_w1 := NOT (NOT #FALSE AND NOT #FALSE) OR #citiTest[4];
   #_w2 := #_w1 AND NOT #citi_Ptrig[4];   // rising edge
   #citi_Ptrig[4] := #_w1;
   "Unit1.ControlNodes".citiMap.PMC.Machining_Assembly.IncrReject_Count := #_w2;
END_REGION

REGION Network 114: Cycle End Trigger 5
   RUNG wire#powerrail
      I_Contact( "Unit1.ControlNodes".citiMap.PMC.Machining_Assembly.IncrGood_Count )
      I_Contact( "Unit1.ControlNodes".citiMap.PMC.Machining_Assembly.IncrReject_Count )
      Not()
      P_Trig( #citi_Ptrig[5] )
      wire#w1
      I_Contact( #citiTon[5].Q )
      Coil( "Unit1.ControlNodes".citiMap.PMC.Machining_Assembly.Cycle_Time_Ready )
   END_RUNG
   RUNG wire#powerrail
      Contact( "Unit1.ControlNodes".citiMap.PMC.Machining_Assembly.Cycle_Time_Ready )
   END_RUNG wire#w1
   RUNG wire#powerrail
      Contact( "Unit1.ControlNodes".citiMap.PMC.Machining_Assembly.Cycle_Time_Ready )
      { S7_Templates := "time_type := Time" } #citiTon[5].TON(pt := #citi, et =>)
   END_RUNG
   // the same network as SCL:
   #_w1 := NOT (NOT "Unit1.ControlNodes".citiMap.PMC.Machining_Assembly.IncrGood_Count AND NOT "Unit1.ControlNodes".citiMap.PMC.Machining_Assembly.IncrReject_Count);
   #_w2 := #_w1 AND NOT #citi_Ptrig[5];   // rising edge
   #citi_Ptrig[5] := #_w1;
   "Unit1.ControlNodes".citiMap.PMC.Machining_Assembly.Cycle_Time_Ready := (#_w2 OR "Unit1.ControlNodes".citiMap.PMC.Machining_Assembly.Cycle_Time_Ready) AND NOT #citiTon[5].Q;
   #citiTon[5].TON(IN := "Unit1.ControlNodes".citiMap.PMC.Machining_Assembly.Cycle_Time_Ready, PT := #citi);
END_REGION

REGION Network 115: Fault bit Level1 6
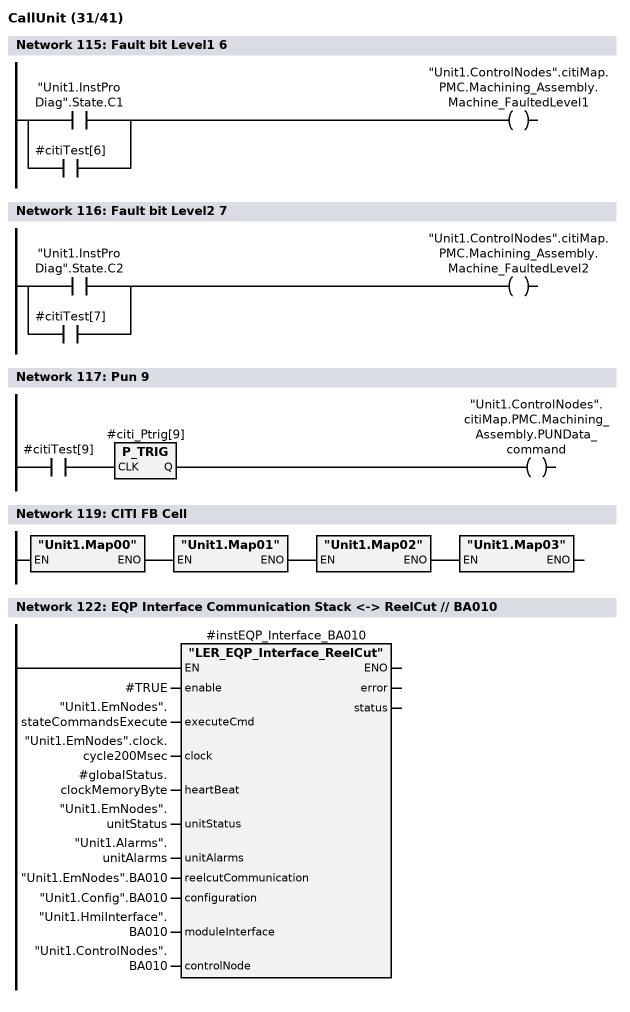
   RUNG wire#powerrail
      Contact( "Unit1.InstProDiag".State.C1 )
      wire#w1
      Coil( "Unit1.ControlNodes".citiMap.PMC.Machining_Assembly.Machine_FaultedLevel1 )
   END_RUNG
   RUNG wire#powerrail
      Contact( #citiTest[6] )
   END_RUNG wire#w1
   // the same network as SCL:
   "Unit1.ControlNodes".citiMap.PMC.Machining_Assembly.Machine_FaultedLevel1 := "Unit1.InstProDiag".State.C1 OR #citiTest[6];
END_REGION

REGION Network 116: Fault bit Level2 7
   RUNG wire#powerrail
      Contact( "Unit1.InstProDiag".State.C2 )
      wire#w1
      Coil( "Unit1.ControlNodes".citiMap.PMC.Machining_Assembly.Machine_FaultedLevel2 )
   END_RUNG
   RUNG wire#powerrail
      Contact( #citiTest[7] )
   END_RUNG wire#w1
   // the same network as SCL:
   "Unit1.ControlNodes".citiMap.PMC.Machining_Assembly.Machine_FaultedLevel2 := "Unit1.InstProDiag".State.C2 OR #citiTest[7];
END_REGION

REGION Network 117: Pun 9
   RUNG wire#powerrail
      Contact( #citiTest[9] )
      P_Trig( #citi_Ptrig[9] )
      Coil( "Unit1.ControlNodes".citiMap.PMC.Machining_Assembly.PUNData_command )
   END_RUNG
   // the same network as SCL:
   #_w1 := #citiTest[9] AND NOT #citi_Ptrig[9];   // rising edge
   #citi_Ptrig[9] := #citiTest[9];
   "Unit1.ControlNodes".citiMap.PMC.Machining_Assembly.PUNData_command := #_w1;
END_REGION

REGION Network 118: ControlNodes.CitiMap -> Unit1. EmNodes.Andon X
END_REGION

REGION Network 119: CITI FB Cell
   RUNG wire#powerrail
      "Unit1.Map00"()
      "Unit1.Map01"()
      "Unit1.Map02"()
      "Unit1.Map03"()
   END_RUNG
   // the same network as SCL:
   "Unit1.Map00"(ENO => #_w1);
   "Unit1.Map01"(EN := #_w1, ENO => #_w2);
   "Unit1.Map02"(EN := #_w2, ENO => #_w3);
   IF #_w3 THEN "Unit1.Map03"(); END_IF;
END_REGION

REGION Network 121: ******************** PLC Communication ********************
END_REGION

REGION Network 122: EQP Interface Communication Stack <-> ReelCut // BA010
   RUNG wire#powerrail
      #instEQP_Interface_BA010(enable := #TRUE, executeCmd := "Unit1.EmNodes".stateCommandsExecute, clock := "Unit1.EmNodes".clock.cycle200Msec, heartBeat := #globalStatus.clockMemoryByte, unitStatus := "Unit1.EmNodes".unitStatus, unitAlarms := "Unit1.Alarms".unitAlarms, reelcutCommunication := "Unit1.EmNodes".BA010, configuration := "Unit1.Config".BA010, moduleInterface := "Unit1.HmiInterface".BA010, controlNode := "Unit1.ControlNodes".BA010, error =>, status =>)
   END_RUNG
   // the same network as SCL:
   #instEQP_Interface_BA010(enable := #TRUE,   // "LER_EQP_Interface_ReelCut"
                           executeCmd := "Unit1.EmNodes".stateCommandsExecute,
                           clock := "Unit1.EmNodes".clock.cycle200Msec,
                           heartBeat := #globalStatus.clockMemoryByte,
                           unitStatus := "Unit1.EmNodes".unitStatus,
                           unitAlarms := "Unit1.Alarms".unitAlarms,
                           reelcutCommunication := "Unit1.EmNodes".BA010,
                           configuration := "Unit1.Config".BA010,
                           moduleInterface := "Unit1.HmiInterface".BA010,
                           controlNode := "Unit1.ControlNodes".BA010);
END_REGION

REGION Network 123: EQP Interface Communication Stack <-> ReelCut // BA015
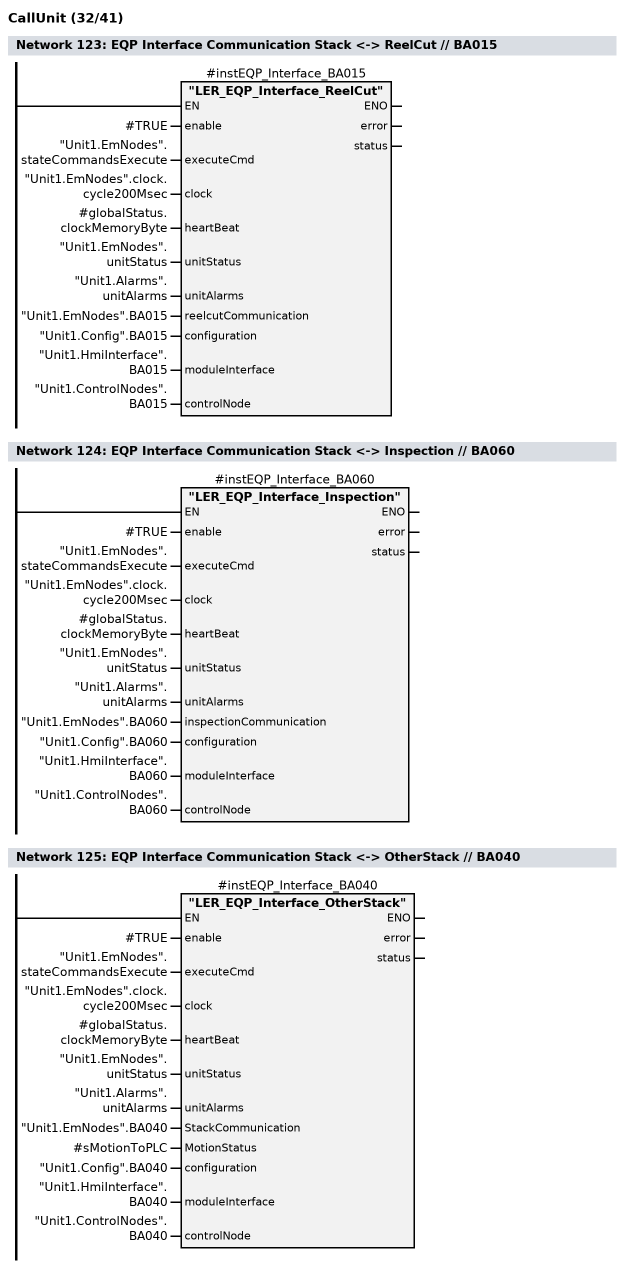
   RUNG wire#powerrail
      #instEQP_Interface_BA015(enable := #TRUE, executeCmd := "Unit1.EmNodes".stateCommandsExecute, clock := "Unit1.EmNodes".clock.cycle200Msec, heartBeat := #globalStatus.clockMemoryByte, unitStatus := "Unit1.EmNodes".unitStatus, unitAlarms := "Unit1.Alarms".unitAlarms, reelcutCommunication := "Unit1.EmNodes".BA015, configuration := "Unit1.Config".BA015, moduleInterface := "Unit1.HmiInterface".BA015, controlNode := "Unit1.ControlNodes".BA015, error =>, status =>)
   END_RUNG
   // the same network as SCL:
   #instEQP_Interface_BA015(enable := #TRUE,   // "LER_EQP_Interface_ReelCut"
                           executeCmd := "Unit1.EmNodes".stateCommandsExecute,
                           clock := "Unit1.EmNodes".clock.cycle200Msec,
                           heartBeat := #globalStatus.clockMemoryByte,
                           unitStatus := "Unit1.EmNodes".unitStatus,
                           unitAlarms := "Unit1.Alarms".unitAlarms,
                           reelcutCommunication := "Unit1.EmNodes".BA015,
                           configuration := "Unit1.Config".BA015,
                           moduleInterface := "Unit1.HmiInterface".BA015,
                           controlNode := "Unit1.ControlNodes".BA015);
END_REGION

REGION Network 124: EQP Interface Communication Stack <-> Inspection // BA060
   RUNG wire#powerrail
      #instEQP_Interface_BA060(enable := #TRUE, executeCmd := "Unit1.EmNodes".stateCommandsExecute, clock := "Unit1.EmNodes".clock.cycle200Msec, heartBeat := #globalStatus.clockMemoryByte, unitStatus := "Unit1.EmNodes".unitStatus, unitAlarms := "Unit1.Alarms".unitAlarms, inspectionCommunication := "Unit1.EmNodes".BA060, configuration := "Unit1.Config".BA060, moduleInterface := "Unit1.HmiInterface".BA060, controlNode := "Unit1.ControlNodes".BA060, error =>, status =>)
   END_RUNG
   // the same network as SCL:
   #instEQP_Interface_BA060(enable := #TRUE,   // "LER_EQP_Interface_Inspection"
                           executeCmd := "Unit1.EmNodes".stateCommandsExecute,
                           clock := "Unit1.EmNodes".clock.cycle200Msec,
                           heartBeat := #globalStatus.clockMemoryByte,
                           unitStatus := "Unit1.EmNodes".unitStatus,
                           unitAlarms := "Unit1.Alarms".unitAlarms,
                           inspectionCommunication := "Unit1.EmNodes".BA060,
                           configuration := "Unit1.Config".BA060,
                           moduleInterface := "Unit1.HmiInterface".BA060,
                           controlNode := "Unit1.ControlNodes".BA060);
END_REGION

REGION Network 125: EQP Interface Communication Stack <-> OtherStack // BA040
   RUNG wire#powerrail
      #instEQP_Interface_BA040(enable := #TRUE, executeCmd := "Unit1.EmNodes".stateCommandsExecute, clock := "Unit1.EmNodes".clock.cycle200Msec, heartBeat := #globalStatus.clockMemoryByte, unitStatus := "Unit1.EmNodes".unitStatus, unitAlarms := "Unit1.Alarms".unitAlarms, StackCommunication := "Unit1.EmNodes".BA040, MotionStatus := #sMotionToPLC, configuration := "Unit1.Config".BA040, moduleInterface := "Unit1.HmiInterface".BA040, controlNode := "Unit1.ControlNodes".BA040, error =>, status =>)
   END_RUNG
   // the same network as SCL:
   #instEQP_Interface_BA040(enable := #TRUE,   // "LER_EQP_Interface_OtherStack"
                           executeCmd := "Unit1.EmNodes".stateCommandsExecute,
                           clock := "Unit1.EmNodes".clock.cycle200Msec,
                           heartBeat := #globalStatus.clockMemoryByte,
                           unitStatus := "Unit1.EmNodes".unitStatus,
                           unitAlarms := "Unit1.Alarms".unitAlarms,
                           StackCommunication := "Unit1.EmNodes".BA040,
                           MotionStatus := #sMotionToPLC,
                           configuration := "Unit1.Config".BA040,
                           moduleInterface := "Unit1.HmiInterface".BA040,
                           controlNode := "Unit1.ControlNodes".BA040);
END_REGION

REGION Network 126: Stack to Reelcut BA10 PackML State
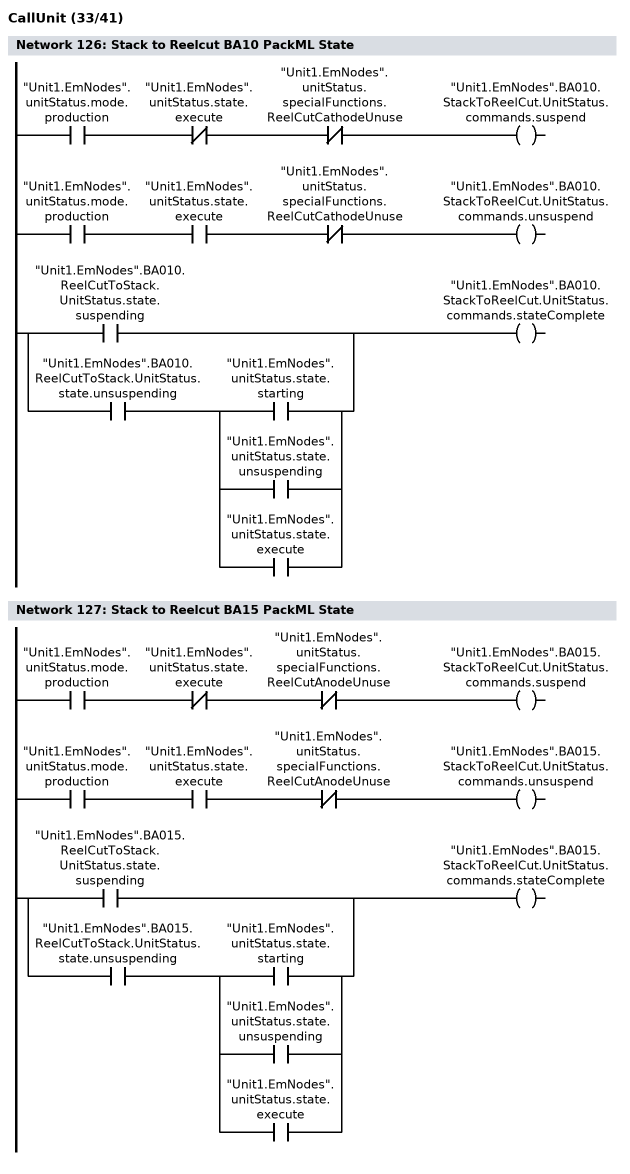
   RUNG wire#powerrail
      Contact( "Unit1.EmNodes".unitStatus.mode.production )
      I_Contact( "Unit1.EmNodes".unitStatus.state.execute )
      I_Contact( "Unit1.EmNodes".unitStatus.specialFunctions.ReelCutCathodeUnuse )
      Coil( "Unit1.EmNodes".BA010.StackToReelCut.UnitStatus.commands.suspend )
   END_RUNG
   RUNG wire#powerrail
      Contact( "Unit1.EmNodes".unitStatus.mode.production )
      Contact( "Unit1.EmNodes".unitStatus.state.execute )
      I_Contact( "Unit1.EmNodes".unitStatus.specialFunctions.ReelCutCathodeUnuse )
      Coil( "Unit1.EmNodes".BA010.StackToReelCut.UnitStatus.commands.unsuspend )
   END_RUNG
   RUNG wire#powerrail
      Contact( "Unit1.EmNodes".BA010.ReelCutToStack.UnitStatus.state.suspending )
      wire#w1
      Coil( "Unit1.EmNodes".BA010.StackToReelCut.UnitStatus.commands.stateComplete )
   END_RUNG
   RUNG wire#powerrail
      Contact( "Unit1.EmNodes".BA010.ReelCutToStack.UnitStatus.state.unsuspending )
      wire#w2
      Contact( "Unit1.EmNodes".unitStatus.state.starting )
   END_RUNG wire#w1
   RUNG wire#w2
      Contact( "Unit1.EmNodes".unitStatus.state.unsuspending )
   END_RUNG wire#w1
   RUNG wire#w2
      Contact( "Unit1.EmNodes".unitStatus.state.execute )
   END_RUNG wire#w1
   // the same network as SCL:
   "Unit1.EmNodes".BA010.StackToReelCut.UnitStatus.commands.suspend := "Unit1.EmNodes".unitStatus.mode.production AND NOT "Unit1.EmNodes".unitStatus.state.execute AND NOT "Unit1.EmNodes".unitStatus.specialFunctions.ReelCutCathodeUnuse;
   "Unit1.EmNodes".BA010.StackToReelCut.UnitStatus.commands.unsuspend := "Unit1.EmNodes".unitStatus.mode.production AND "Unit1.EmNodes".unitStatus.state.execute AND NOT "Unit1.EmNodes".unitStatus.specialFunctions.ReelCutCathodeUnuse;
   "Unit1.EmNodes".BA010.StackToReelCut.UnitStatus.commands.stateComplete := "Unit1.EmNodes".BA010.ReelCutToStack.UnitStatus.state.suspending OR ("Unit1.EmNodes".BA010.ReelCutToStack.UnitStatus.state.unsuspending AND ("Unit1.EmNodes".unitStatus.state.starting OR "Unit1.EmNodes".unitStatus.state.unsuspending OR "Unit1.EmNodes".unitStatus.state.execute));
END_REGION

REGION Network 127: Stack to Reelcut BA15 PackML State
   RUNG wire#powerrail
      Contact( "Unit1.EmNodes".unitStatus.mode.production )
      I_Contact( "Unit1.EmNodes".unitStatus.state.execute )
      I_Contact( "Unit1.EmNodes".unitStatus.specialFunctions.ReelCutAnodeUnuse )
      Coil( "Unit1.EmNodes".BA015.StackToReelCut.UnitStatus.commands.suspend )
   END_RUNG
   RUNG wire#powerrail
      Contact( "Unit1.EmNodes".unitStatus.mode.production )
      Contact( "Unit1.EmNodes".unitStatus.state.execute )
      I_Contact( "Unit1.EmNodes".unitStatus.specialFunctions.ReelCutAnodeUnuse )
      Coil( "Unit1.EmNodes".BA015.StackToReelCut.UnitStatus.commands.unsuspend )
   END_RUNG
   RUNG wire#powerrail
      Contact( "Unit1.EmNodes".BA015.ReelCutToStack.UnitStatus.state.suspending )
      wire#w1
      Coil( "Unit1.EmNodes".BA015.StackToReelCut.UnitStatus.commands.stateComplete )
   END_RUNG
   RUNG wire#powerrail
      Contact( "Unit1.EmNodes".BA015.ReelCutToStack.UnitStatus.state.unsuspending )
      wire#w2
      Contact( "Unit1.EmNodes".unitStatus.state.starting )
   END_RUNG wire#w1
   RUNG wire#w2
      Contact( "Unit1.EmNodes".unitStatus.state.unsuspending )
   END_RUNG wire#w1
   RUNG wire#w2
      Contact( "Unit1.EmNodes".unitStatus.state.execute )
   END_RUNG wire#w1
   // the same network as SCL:
   "Unit1.EmNodes".BA015.StackToReelCut.UnitStatus.commands.suspend := "Unit1.EmNodes".unitStatus.mode.production AND NOT "Unit1.EmNodes".unitStatus.state.execute AND NOT "Unit1.EmNodes".unitStatus.specialFunctions.ReelCutAnodeUnuse;
   "Unit1.EmNodes".BA015.StackToReelCut.UnitStatus.commands.unsuspend := "Unit1.EmNodes".unitStatus.mode.production AND "Unit1.EmNodes".unitStatus.state.execute AND NOT "Unit1.EmNodes".unitStatus.specialFunctions.ReelCutAnodeUnuse;
   "Unit1.EmNodes".BA015.StackToReelCut.UnitStatus.commands.stateComplete := "Unit1.EmNodes".BA015.ReelCutToStack.UnitStatus.state.suspending OR ("Unit1.EmNodes".BA015.ReelCutToStack.UnitStatus.state.unsuspending AND ("Unit1.EmNodes".unitStatus.state.starting OR "Unit1.EmNodes".unitStatus.state.unsuspending OR "Unit1.EmNodes".unitStatus.state.execute));
END_REGION

REGION Network 128: Stack to Reelcut BA60 PackML State
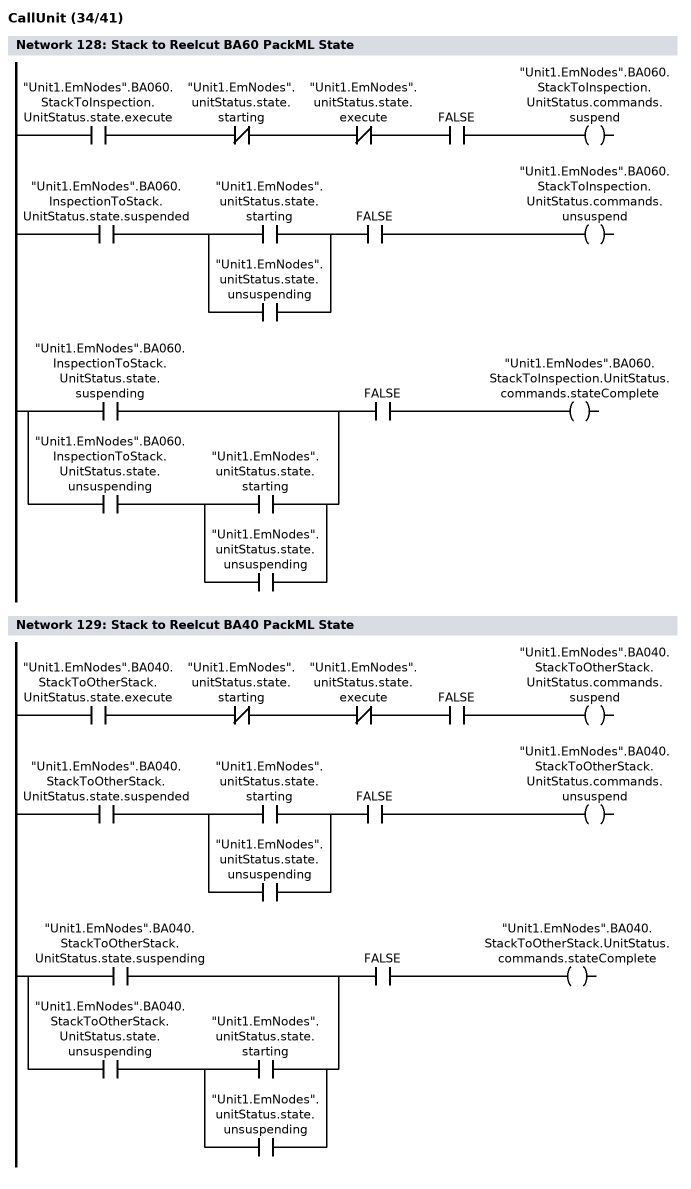
   RUNG wire#powerrail
      Contact( "Unit1.EmNodes".BA060.StackToInspection.UnitStatus.state.execute )
      I_Contact( "Unit1.EmNodes".unitStatus.state.starting )
      I_Contact( "Unit1.EmNodes".unitStatus.state.execute )
      Contact( FALSE )
      Coil( "Unit1.EmNodes".BA060.StackToInspection.UnitStatus.commands.suspend )
   END_RUNG
   RUNG wire#powerrail
      Contact( "Unit1.EmNodes".BA060.InspectionToStack.UnitStatus.state.suspended )
      wire#w1
      Contact( "Unit1.EmNodes".unitStatus.state.starting )
      wire#w2
      Contact( FALSE )
      Coil( "Unit1.EmNodes".BA060.StackToInspection.UnitStatus.commands.unsuspend )
   END_RUNG
   RUNG wire#w1
      Contact( "Unit1.EmNodes".unitStatus.state.unsuspending )
   END_RUNG wire#w2
   RUNG wire#powerrail
      Contact( "Unit1.EmNodes".BA060.InspectionToStack.UnitStatus.state.suspending )
      wire#w3
      Contact( FALSE )
      Coil( "Unit1.EmNodes".BA060.StackToInspection.UnitStatus.commands.stateComplete )
   END_RUNG
   RUNG wire#powerrail
      Contact( "Unit1.EmNodes".BA060.InspectionToStack.UnitStatus.state.unsuspending )
      wire#w4
      Contact( "Unit1.EmNodes".unitStatus.state.starting )
   END_RUNG wire#w3
   RUNG wire#w4
      Contact( "Unit1.EmNodes".unitStatus.state.unsuspending )
   END_RUNG wire#w3
   // the same network as SCL:
   "Unit1.EmNodes".BA060.StackToInspection.UnitStatus.commands.suspend := "Unit1.EmNodes".BA060.StackToInspection.UnitStatus.state.execute AND NOT "Unit1.EmNodes".unitStatus.state.starting AND NOT "Unit1.EmNodes".unitStatus.state.execute AND FALSE;
   "Unit1.EmNodes".BA060.StackToInspection.UnitStatus.commands.unsuspend := "Unit1.EmNodes".BA060.InspectionToStack.UnitStatus.state.suspended AND ("Unit1.EmNodes".unitStatus.state.starting OR "Unit1.EmNodes".unitStatus.state.unsuspending) AND FALSE;
   "Unit1.EmNodes".BA060.StackToInspection.UnitStatus.commands.stateComplete := ("Unit1.EmNodes".BA060.InspectionToStack.UnitStatus.state.suspending OR ("Unit1.EmNodes".BA060.InspectionToStack.UnitStatus.state.unsuspending AND ("Unit1.EmNodes".unitStatus.state.starting OR "Unit1.EmNodes".unitStatus.state.unsuspending))) AND FALSE;
END_REGION

REGION Network 129: Stack to Reelcut BA40 PackML State
   RUNG wire#powerrail
      Contact( "Unit1.EmNodes".BA040.StackToOtherStack.UnitStatus.state.execute )
      I_Contact( "Unit1.EmNodes".unitStatus.state.starting )
      I_Contact( "Unit1.EmNodes".unitStatus.state.execute )
      Contact( FALSE )
      Coil( "Unit1.EmNodes".BA040.StackToOtherStack.UnitStatus.commands.suspend )
   END_RUNG
   RUNG wire#powerrail
      Contact( "Unit1.EmNodes".BA040.StackToOtherStack.UnitStatus.state.suspended )
      wire#w1
      Contact( "Unit1.EmNodes".unitStatus.state.starting )
      wire#w2
      Contact( FALSE )
      Coil( "Unit1.EmNodes".BA040.StackToOtherStack.UnitStatus.commands.unsuspend )
   END_RUNG
   RUNG wire#w1
      Contact( "Unit1.EmNodes".unitStatus.state.unsuspending )
   END_RUNG wire#w2
   RUNG wire#powerrail
      Contact( "Unit1.EmNodes".BA040.StackToOtherStack.UnitStatus.state.suspending )
      wire#w3
      Contact( FALSE )
      Coil( "Unit1.EmNodes".BA040.StackToOtherStack.UnitStatus.commands.stateComplete )
   END_RUNG
   RUNG wire#powerrail
      Contact( "Unit1.EmNodes".BA040.StackToOtherStack.UnitStatus.state.unsuspending )
      wire#w4
      Contact( "Unit1.EmNodes".unitStatus.state.starting )
   END_RUNG wire#w3
   RUNG wire#w4
      Contact( "Unit1.EmNodes".unitStatus.state.unsuspending )
   END_RUNG wire#w3
   // the same network as SCL:
   "Unit1.EmNodes".BA040.StackToOtherStack.UnitStatus.commands.suspend := "Unit1.EmNodes".BA040.StackToOtherStack.UnitStatus.state.execute AND NOT "Unit1.EmNodes".unitStatus.state.starting AND NOT "Unit1.EmNodes".unitStatus.state.execute AND FALSE;
   "Unit1.EmNodes".BA040.StackToOtherStack.UnitStatus.commands.unsuspend := "Unit1.EmNodes".BA040.StackToOtherStack.UnitStatus.state.suspended AND ("Unit1.EmNodes".unitStatus.state.starting OR "Unit1.EmNodes".unitStatus.state.unsuspending) AND FALSE;
   "Unit1.EmNodes".BA040.StackToOtherStack.UnitStatus.commands.stateComplete := ("Unit1.EmNodes".BA040.StackToOtherStack.UnitStatus.state.suspending OR ("Unit1.EmNodes".BA040.StackToOtherStack.UnitStatus.state.unsuspending AND ("Unit1.EmNodes".unitStatus.state.starting OR "Unit1.EmNodes".unitStatus.state.unsuspending))) AND FALSE;
END_REGION

REGION Network 130: BA010 Interface Data
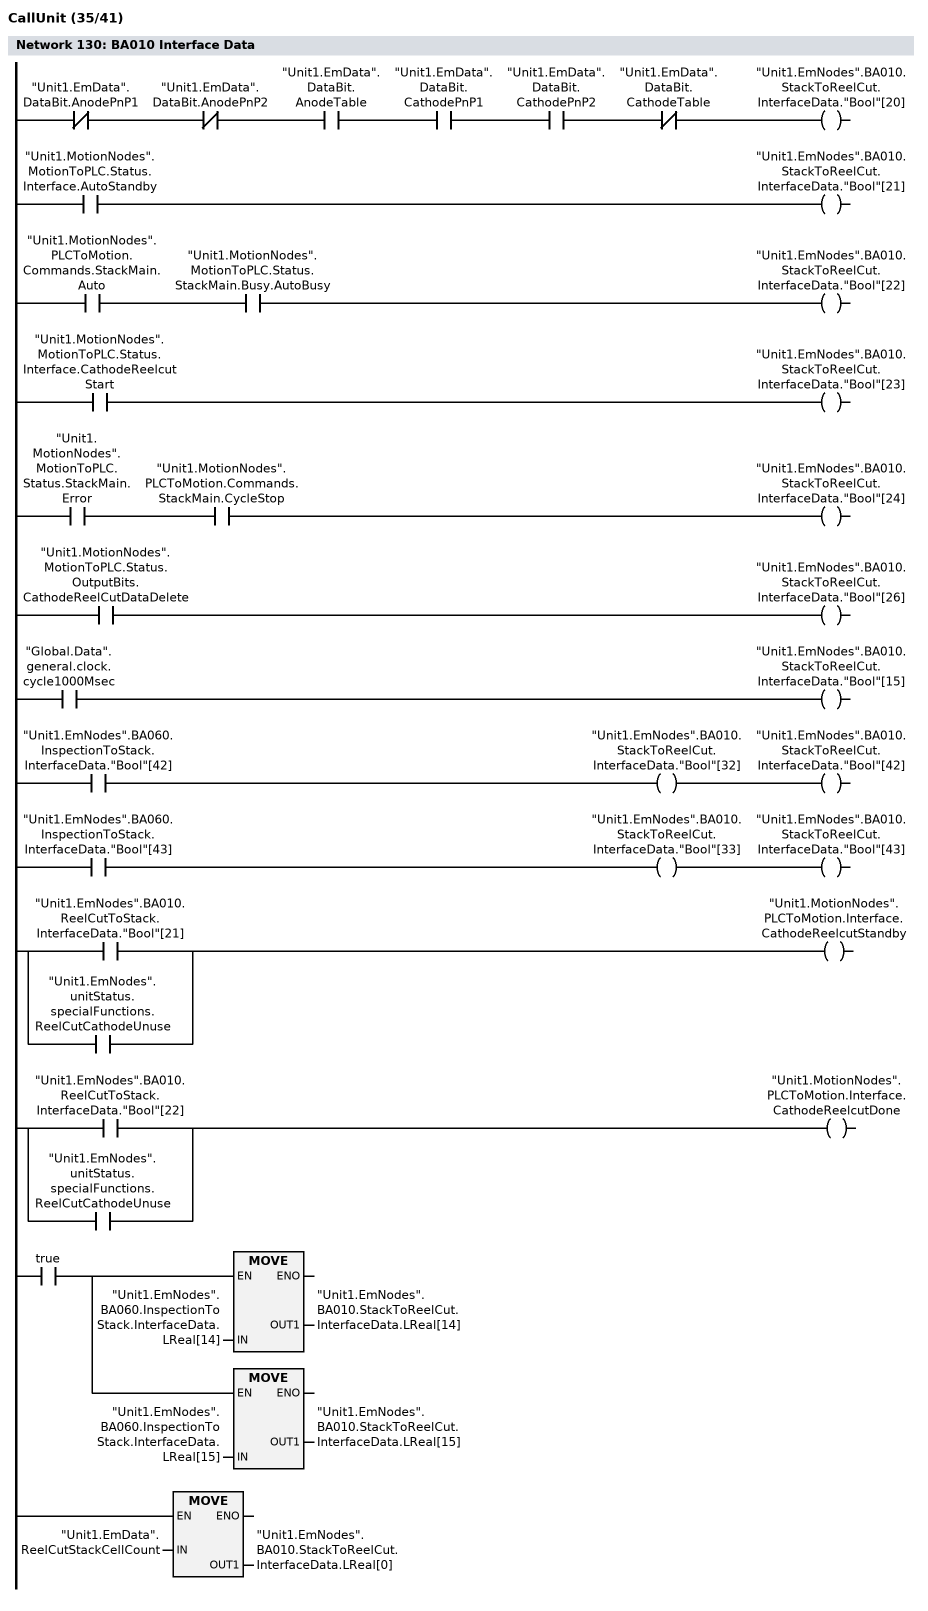
   RUNG wire#powerrail
      I_Contact( "Unit1.EmData".DataBit.AnodePnP1 )
      I_Contact( "Unit1.EmData".DataBit.AnodePnP2 )
      Contact( "Unit1.EmData".DataBit.AnodeTable )
      Contact( "Unit1.EmData".DataBit.CathodePnP1 )
      Contact( "Unit1.EmData".DataBit.CathodePnP2 )
      I_Contact( "Unit1.EmData".DataBit.CathodeTable )
      Coil( "Unit1.EmNodes".BA010.StackToReelCut.InterfaceData."Bool"[20] )
   END_RUNG
   RUNG wire#powerrail
      Contact( "Unit1.MotionNodes".MotionToPLC.Status.Interface.AutoStandby )
      Coil( "Unit1.EmNodes".BA010.StackToReelCut.InterfaceData."Bool"[21] )
   END_RUNG
   RUNG wire#powerrail
      Contact( "Unit1.MotionNodes".PLCToMotion.Commands.StackMain.Auto )
      Contact( "Unit1.MotionNodes".MotionToPLC.Status.StackMain.Busy.AutoBusy )
      Coil( "Unit1.EmNodes".BA010.StackToReelCut.InterfaceData."Bool"[22] )
   END_RUNG
   RUNG wire#powerrail
      Contact( "Unit1.MotionNodes".MotionToPLC.Status.Interface.CathodeReelcutStart )
      Coil( "Unit1.EmNodes".BA010.StackToReelCut.InterfaceData."Bool"[23] )
   END_RUNG
   RUNG wire#powerrail
      Contact( "Unit1.MotionNodes".MotionToPLC.Status.StackMain.Error )
      Contact( "Unit1.MotionNodes".PLCToMotion.Commands.StackMain.CycleStop )
      Coil( "Unit1.EmNodes".BA010.StackToReelCut.InterfaceData."Bool"[24] )
   END_RUNG
   RUNG wire#powerrail
      Contact( "Unit1.MotionNodes".MotionToPLC.Status.OutputBits.CathodeReelCutDataDelete )
      Coil( "Unit1.EmNodes".BA010.StackToReelCut.InterfaceData."Bool"[26] )
   END_RUNG
   RUNG wire#powerrail
      Contact( "Global.Data".general.clock.cycle1000Msec )
      Coil( "Unit1.EmNodes".BA010.StackToReelCut.InterfaceData."Bool"[15] )
   END_RUNG
   RUNG wire#powerrail
      Contact( "Unit1.EmNodes".BA060.InspectionToStack.InterfaceData."Bool"[42] )
      Coil( "Unit1.EmNodes".BA010.StackToReelCut.InterfaceData."Bool"[32] )
      Coil( "Unit1.EmNodes".BA010.StackToReelCut.InterfaceData."Bool"[42] )
   END_RUNG
   RUNG wire#powerrail
      Contact( "Unit1.EmNodes".BA060.InspectionToStack.InterfaceData."Bool"[43] )
      Coil( "Unit1.EmNodes".BA010.StackToReelCut.InterfaceData."Bool"[33] )
      Coil( "Unit1.EmNodes".BA010.StackToReelCut.InterfaceData."Bool"[43] )
   END_RUNG
   RUNG wire#powerrail
      Contact( "Unit1.EmNodes".BA010.ReelCutToStack.InterfaceData."Bool"[21] )
      wire#w1
      Coil( "Unit1.MotionNodes".PLCToMotion.Interface.CathodeReelcutStandby )
   END_RUNG
   RUNG wire#powerrail
      Contact( "Unit1.EmNodes".unitStatus.specialFunctions.ReelCutCathodeUnuse )
   END_RUNG wire#w1
   RUNG wire#powerrail
      Contact( "Unit1.EmNodes".BA010.ReelCutToStack.InterfaceData."Bool"[22] )
      wire#w2
      Coil( "Unit1.MotionNodes".PLCToMotion.Interface.CathodeReelcutDone )
   END_RUNG
   RUNG wire#powerrail
      Contact( "Unit1.EmNodes".unitStatus.specialFunctions.ReelCutCathodeUnuse )
   END_RUNG wire#w2
   RUNG wire#powerrail
      Contact( true )
      wire#w3
      Move(in := "Unit1.EmNodes".BA060.InspectionToStack.InterfaceData.LReal[14], out1 => "Unit1.EmNodes".BA010.StackToReelCut.InterfaceData.LReal[14])
   END_RUNG
   RUNG wire#w3
      Move(in := "Unit1.EmNodes".BA060.InspectionToStack.InterfaceData.LReal[15], out1 => "Unit1.EmNodes".BA010.StackToReelCut.InterfaceData.LReal[15])
   END_RUNG
   RUNG wire#powerrail
      Move(in := "Unit1.EmData".ReelCutStackCellCount, out1 => "Unit1.EmNodes".BA010.StackToReelCut.InterfaceData.LReal[0])
   END_RUNG
   // the same network as SCL:
   "Unit1.EmNodes".BA010.StackToReelCut.InterfaceData."Bool"[20] := NOT "Unit1.EmData".DataBit.AnodePnP1 AND NOT "Unit1.EmData".DataBit.AnodePnP2 AND "Unit1.EmData".DataBit.AnodeTable AND "Unit1.EmData".DataBit.CathodePnP1 AND "Unit1.EmData".DataBit.CathodePnP2 AND NOT "Unit1.EmData".DataBit.CathodeTable;
   "Unit1.EmNodes".BA010.StackToReelCut.InterfaceData."Bool"[21] := "Unit1.MotionNodes".MotionToPLC.Status.Interface.AutoStandby;
   "Unit1.EmNodes".BA010.StackToReelCut.InterfaceData."Bool"[22] := "Unit1.MotionNodes".PLCToMotion.Commands.StackMain.Auto AND "Unit1.MotionNodes".MotionToPLC.Status.StackMain.Busy.AutoBusy;
   "Unit1.EmNodes".BA010.StackToReelCut.InterfaceData."Bool"[23] := "Unit1.MotionNodes".MotionToPLC.Status.Interface.CathodeReelcutStart;
   "Unit1.EmNodes".BA010.StackToReelCut.InterfaceData."Bool"[24] := "Unit1.MotionNodes".MotionToPLC.Status.StackMain.Error AND "Unit1.MotionNodes".PLCToMotion.Commands.StackMain.CycleStop;
   "Unit1.EmNodes".BA010.StackToReelCut.InterfaceData."Bool"[26] := "Unit1.MotionNodes".MotionToPLC.Status.OutputBits.CathodeReelCutDataDelete;
   "Unit1.EmNodes".BA010.StackToReelCut.InterfaceData."Bool"[15] := "Global.Data".general.clock.cycle1000Msec;
   "Unit1.EmNodes".BA010.StackToReelCut.InterfaceData."Bool"[32] := "Unit1.EmNodes".BA060.InspectionToStack.InterfaceData."Bool"[42];
   "Unit1.EmNodes".BA010.StackToReelCut.InterfaceData."Bool"[42] := "Unit1.EmNodes".BA060.InspectionToStack.InterfaceData."Bool"[42];
   "Unit1.EmNodes".BA010.StackToReelCut.InterfaceData."Bool"[33] := "Unit1.EmNodes".BA060.InspectionToStack.InterfaceData."Bool"[43];
   "Unit1.EmNodes".BA010.StackToReelCut.InterfaceData."Bool"[43] := "Unit1.EmNodes".BA060.InspectionToStack.InterfaceData."Bool"[43];
   "Unit1.MotionNodes".PLCToMotion.Interface.CathodeReelcutStandby := "Unit1.EmNodes".BA010.ReelCutToStack.InterfaceData."Bool"[21] OR "Unit1.EmNodes".unitStatus.specialFunctions.ReelCutCathodeUnuse;
   "Unit1.MotionNodes".PLCToMotion.Interface.CathodeReelcutDone := "Unit1.EmNodes".BA010.ReelCutToStack.InterfaceData."Bool"[22] OR "Unit1.EmNodes".unitStatus.specialFunctions.ReelCutCathodeUnuse;
   IF true THEN
       "Unit1.EmNodes".BA010.StackToReelCut.InterfaceData.LReal[14] := "Unit1.EmNodes".BA060.InspectionToStack.InterfaceData.LReal[14];
       "Unit1.EmNodes".BA010.StackToReelCut.InterfaceData.LReal[15] := "Unit1.EmNodes".BA060.InspectionToStack.InterfaceData.LReal[15];
   END_IF;
   "Unit1.EmNodes".BA010.StackToReelCut.InterfaceData.LReal[0] := "Unit1.EmData".ReelCutStackCellCount;
END_REGION

REGION Network 131: Stack To ReelCut BA010 Unit Status
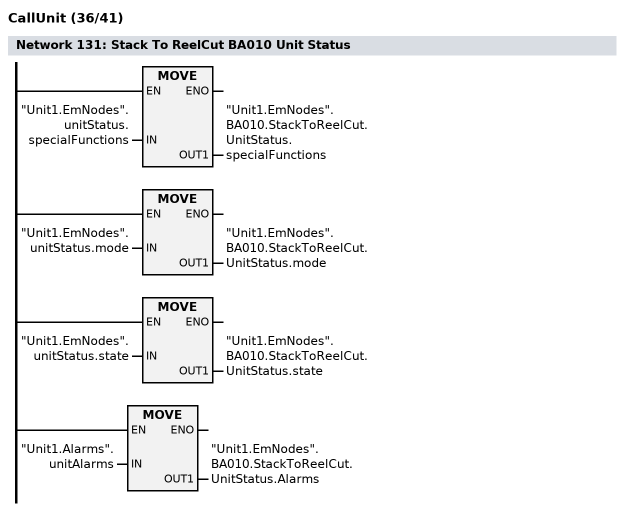
   RUNG wire#powerrail
      Move(in := "Unit1.EmNodes".unitStatus.specialFunctions, out1 => "Unit1.EmNodes".BA010.StackToReelCut.UnitStatus.specialFunctions)
   END_RUNG
   RUNG wire#powerrail
      Move(in := "Unit1.EmNodes".unitStatus.mode, out1 => "Unit1.EmNodes".BA010.StackToReelCut.UnitStatus.mode)
   END_RUNG
   RUNG wire#powerrail
      Move(in := "Unit1.EmNodes".unitStatus.state, out1 => "Unit1.EmNodes".BA010.StackToReelCut.UnitStatus.state)
   END_RUNG
   RUNG wire#powerrail
      Move(in := "Unit1.Alarms".unitAlarms, out1 => "Unit1.EmNodes".BA010.StackToReelCut.UnitStatus.Alarms)
   END_RUNG
   // the same network as SCL:
   "Unit1.EmNodes".BA010.StackToReelCut.UnitStatus.specialFunctions := "Unit1.EmNodes".unitStatus.specialFunctions;
   "Unit1.EmNodes".BA010.StackToReelCut.UnitStatus.mode := "Unit1.EmNodes".unitStatus.mode;
   "Unit1.EmNodes".BA010.StackToReelCut.UnitStatus.state := "Unit1.EmNodes".unitStatus.state;
   "Unit1.EmNodes".BA010.StackToReelCut.UnitStatus.Alarms := "Unit1.Alarms".unitAlarms;
END_REGION

